LIN {X 0,Y 171.052,Z 952.165,A -85,B 0,C 180,E1 8008.321,E2 8008.321} C_VEL
LIN {X 0,Y 174.911,Z 942.549,A -85,B 0,C 180,E1 8004.093,E2 8004.093} C_VEL
LIN {X 0,Y 179.129,Z 931.53,A -85,B 0,C 180,E1 8000.36,E2 8000.36} C_VEL
LIN {X 0,Y 183.775,Z 918.134,A -85,B 0,C 180,E1 7996.88,E2 7996.88} C_VEL
LIN {X 0,Y 187.844,Z 904.879,A -85,B 0,C 180,E1 7994.248,E2 7994.248} C_VEL
LIN {X 0,Y 191.799,Z 889.443,A -85,B 0,C 180,E1 7991.93,E2 7991.93} C_VEL
LIN {X 0,Y 194.927,Z 873.983,A -85,B 0,C 180,E1 7990.211,E2 7990.211} C_VEL
LIN {X 0,Y 197.39,Z 856.631,A -85,B 0,C 180,E1 7988.872,E2 7988.872} C_VEL
LIN {X 0,Y 198.822,Z 839.35,A -85,B 0,C 180,E1 7988.05,E2 7988.05} C_VEL
LIN {X 0,Y 203.826,Z 763.58,A -85,B 0,C 180,E1 7985.576,E2 7985.576} C_VEL
LIN {X 0,Y 200.047,Z 723.867,A -85,B 0,C 180,E1 7982.552,E2 7982.552} C_VEL
LIN {X 0,Y 192.576,Z 708.428,A -85,B 0,C 180,E1 7979.398,E2 7979.398} C_VEL
LIN {X 0,Y 189.739,Z 703.046,A -85,B 0,C 180,E1 7978.041,E2 7978.041} C_VEL
LIN {X 0,Y 187.484,Z 693.288,A -85,B 0,C 180,E1 7973.127,E2 7973.127} C_VEL
LIN {X 0,Y 185.114,Z 684.758,A -85,B 0,C 180,E1 7967.95,E2 7967.95} C_VEL
LIN {X 0,Y 182.975,Z 677.799,A -85,B 0,C 180,E1 7962.924,E2 7962.924} C_VEL
LIN {X 0,Y 180.958,Z 671.792,A -85,B 0,C 180,E1 7957.631,E2 7957.631} C_VEL
LIN {X 0,Y 179.391,Z 667.819,A -85,B 0,C 180,E1 7953.109,E2 7953.109} C_VEL
LIN {X 0,Y 178.095,Z 664.338,A -85,B 0,C 180,E1 7948.138,E2 7948.138} C_VEL
LIN {X 0,Y 176.788,Z 660.79,A -85,B 0,C 180,E1 7939.838,E2 7939.838} C_VEL
LIN {X 0,Y 176.356,Z 660.229,A -85,B 0,C 180,E1 7933.442,E2 7933.442} C_VEL
LIN {X 0,Y 176.924,Z 660.85,A -85,B 0,C 180,E1 7927.143,E2 7927.143} C_VEL
LIN {X 0,Y 177.553,Z 662.846,A -85,B 0,C 180,E1 7922.26,E2 7922.26} C_VEL
LIN {X 0,Y 179.139,Z 665.796,A -85,B 0,C 180,E1 7916.801,E2 7916.801} C_VEL
LIN {X 0,Y 180.896,Z 669.96,A -85,B 0,C 180,E1 7911.738,E2 7911.738} C_VEL
LIN {X 0,Y 182.615,Z 674.195,A -85,B 0,C 180,E1 7907.671,E2 7907.671} C_VEL
LIN {X 0,Y 185.129,Z 680.488,A -85,B 0,C 180,E1 7902.72,E2 7902.72} C_VEL
LIN {X 0,Y 188.226,Z 689.312,A -85,B 0,C 180,E1 7897.184,E2 7897.184} C_VEL
LIN {X 0,Y 191.226,Z 698.648,A -85,B 0,C 180,E1 7892.416,E2 7892.416} C_VEL
LIN {X 0,Y 199.887,Z 713.757,A -85,B 0,C 180,E1 7888.779,E2 7888.779} C_VEL
LIN {X 0,Y 208.278,Z 730.588,A -85,B 0,C 180,E1 7885.621,E2 7885.621} C_VEL
LIN {X 0,Y 209.07,Z 733.001,A -85,B 0,C 180,E1 7885.302,E2 7885.302} C_VEL
LIN {X 0,Y 209.295,Z 744.68,A -85,B 0,C 180,E1 7884.7,E2 7884.7} C_VEL
LIN {X 0,Y 204.046,Z 825.384,A -85,B 0,C 180,E1 7882.3,E2 7882.3} C_VEL
LIN {X 0,Y 202.813,Z 833.052,A -85,B 0,C 180,E1 7882.253,E2 7882.253} C_VEL
LIN {X 0,Y 196.734,Z 853.33,A -85,B 0,C 180,E1 7882.805,E2 7882.805} C_VEL
LIN {X 0,Y 195.772,Z 859.913,A -85,B 0,C 180,E1 7882.739,E2 7882.739} C_VEL
LIN {X 0,Y 194.086,Z 879.533,A -85,B 0,C 180,E1 7881.974,E2 7881.974} C_VEL
LIN {X 0,Y 191.393,Z 896.772,A -85,B 0,C 180,E1 7880.877,E2 7880.877} C_VEL
LIN {X 0,Y 187.689,Z 913.328,A -85,B 0,C 180,E1 7879.389,E2 7879.389} C_VEL
LIN {X 0,Y 183.008,Z 930.142,A -85,B 0,C 180,E1 7877.295,E2 7877.295} C_VEL
LIN {X 0,Y 177.846,Z 945.933,A -85,B 0,C 180,E1 7874.65,E2 7874.65} C_VEL
LIN {X 0,Y 172.438,Z 960.631,A -85,B 0,C 180,E1 7871.378,E2 7871.378} C_VEL
LIN {X 0,Y 167.021,Z 974.241,A -85,B 0,C 180,E1 7867.419,E2 7867.419} C_VEL
LIN {X 0,Y 162.202,Z 986.322,A -85,B 0,C 180,E1 7862.852,E2 7862.852} C_VEL
LIN {X 0,Y 158.332,Z 996.58,A -85,B 0,C 180,E1 7857.861,E2 7857.861} C_VEL
LIN {X 0,Y 155.474,Z 1005.619,A -85,B 0,C 180,E1 7852.171,E2 7852.171} C_VEL
LIN {X 0,Y 154.031,Z 1012.929,A -85,B 0,C 180,E1 7846.116,E2 7846.116} C_VEL
LIN {X 0,Y 154.049,Z 1018.633,A -85,B 0,C 180,E1 7839.716,E2 7839.716} C_VEL
LIN {X 0,Y 155.156,Z 1022.277,A -85,B 0,C 180,E1 7833.696,E2 7833.696} C_VEL
LIN {X 0,Y 155.745,Z 1023.623,A -85,B 0,C 180,E1 7830.001,E2 7830.001} C_VEL
LIN {X 0,Y 154.747,Z 1024.067,A -85,B 0,C 180,E1 7825.554,E2 7825.554} C_VEL
LIN {X 0,Y 153.525,Z 1023.151,A -85,B 0,C 180,E1 7819.114,E2 7819.114} C_VEL
LIN {X 0,Y 153.864,Z 1020.428,A -85,B 0,C 180,E1 7812.217,E2 7812.217} C_VEL
LIN {X 0,Y 156.454,Z 1015.626,A -85,B 0,C 180,E1 7805.053,E2 7805.053} C_VEL
LIN {X 0,Y 161.104,Z 1009.155,A -85,B 0,C 180,E1 7798.579,E2 7798.579} C_VEL
LIN {X 0,Y 167.354,Z 1001.09,A -85,B 0,C 180,E1 7792.885,E2 7792.885} C_VEL
LIN {X 0,Y 174.735,Z 991.559,A -85,B 0,C 180,E1 7787.973,E2 7787.973} C_VEL
LIN {X 0,Y 182.872,Z 980.59,A -85,B 0,C 180,E1 7783.804,E2 7783.804} C_VEL
LIN {X 0,Y 191.37,Z 968.139,A -85,B 0,C 180,E1 7780.288,E2 7780.288} C_VEL
LIN {X 0,Y 199.606,Z 954.564,A -85,B 0,C 180,E1 7777.444,E2 7777.444} C_VEL
LIN {X 0,Y 207.323,Z 939.977,A -85,B 0,C 180,E1 7775.17,E2 7775.17} C_VEL
LIN {X 0,Y 214.323,Z 924.465,A -85,B 0,C 180,E1 7773.377,E2 7773.377} C_VEL
LIN {X 0,Y 220.444,Z 907.954,A -85,B 0,C 180,E1 7771.987,E2 7771.987} C_VEL
LIN {X 0,Y 225.279,Z 890.795,A -85,B 0,C 180,E1 7770.956,E2 7770.956} C_VEL
LIN {X 0,Y 228.713,Z 872.873,A -85,B 0,C 180,E1 7770.206,E2 7770.206} C_VEL
LIN {X 0,Y 231.397,Z 846.525,A -85,B 0,C 180,E1 7769.481,E2 7769.481} C_VEL
LIN {X 0,Y 238.924,Z 762.658,A -85,B 0,C 180,E1 7767.341,E2 7767.341} C_VEL
LIN {X 0,Y 234.578,Z 754.168,A -85,B 0,C 180,E1 7764.153,E2 7764.153} C_VEL
LIN {X 0,Y 231.17,Z 748.178,A -85,B 0,C 180,E1 7761.171,E2 7761.171} C_VEL
LIN {X 0,Y 228.461,Z 743.864,A -85,B 0,C 180,E1 7758.367,E2 7758.367} C_VEL
LIN {X 0,Y 225.969,Z 740.04,A -85,B 0,C 180,E1 7755.001,E2 7755.001} C_VEL
LIN {X 0,Y 223.932,Z 737.117,A -85,B 0,C 180,E1 7751.069,E2 7751.069} C_VEL
LIN {X 0,Y 222.678,Z 736.115,A -85,B 0,C 180,E1 7745.669,E2 7745.669} C_VEL
LIN {X 0,Y 222.804,Z 736.608,A -85,B 0,C 180,E1 7742.572,E2 7742.572} C_VEL
LIN {X 0,Y 224.405,Z 740.091,A -85,B 0,C 180,E1 7737.062,E2 7737.062} C_VEL
LIN {X 0,Y 226.766,Z 744.94,A -85,B 0,C 180,E1 7733.035,E2 7733.035} C_VEL
LIN {X 0,Y 228.583,Z 748.757,A -85,B 0,C 180,E1 7730.686,E2 7730.686} C_VEL
LIN {X 0,Y 231.247,Z 754.355,A -85,B 0,C 180,E1 7727.894,E2 7727.894} C_VEL
LIN {X 0,Y 234.202,Z 761.168,A -85,B 0,C 180,E1 7725.221,E2 7725.221} C_VEL
LIN {X 0,Y 235.779,Z 765.509,A -85,B 0,C 180,E1 7723.904,E2 7723.904} C_VEL
LIN {X 0,Y 236.085,Z 777.578,A -85,B 0,C 180,E1 7722.777,E2 7722.777} C_VEL
LIN {X 0,Y 228.922,Z 852.059,A -85,B 0,C 180,E1 7720.74,E2 7720.74} C_VEL
LIN {X 0,Y 226.241,Z 868.551,A -85,B 0,C 180,E1 7719.928,E2 7719.928} C_VEL
LIN {X 0,Y 222.3,Z 884.631,A -85,B 0,C 180,E1 7718.775,E2 7718.775} C_VEL
LIN {X 0,Y 217.471,Z 899.315,A -85,B 0,C 180,E1 7717.34,E2 7717.34} C_VEL
LIN {X 0,Y 211.583,Z 913.363,A -85,B 0,C 180,E1 7715.509,E2 7715.509} C_VEL
LIN {X 0,Y 204.895,Z 926.51,A -85,B 0,C 180,E1 7713.254,E2 7713.254} C_VEL
LIN {X 0,Y 197.577,Z 938.587,A -85,B 0,C 180,E1 7710.507,E2 7710.507} C_VEL
LIN {X 0,Y 190.099,Z 949.092,A -85,B 0,C 180,E1 7707.304,E2 7707.304} C_VEL
LIN {X 0,Y 182.682,Z 958.18,A -85,B 0,C 180,E1 7703.568,E2 7703.568} C_VEL
LIN {X 0,Y 175.545,Z 965.705,A -85,B 0,C 180,E1 7699.247,E2 7699.247} C_VEL
LIN {X 0,Y 169.015,Z 971.648,A -85,B 0,C 180,E1 7694.271,E2 7694.271} C_VEL
LIN {X 0,Y 163.752,Z 975.649,A -85,B 0,C 180,E1 7688.969,E2 7688.969} C_VEL
LIN {X 0,Y 159.527,Z 977.967,A -85,B 0,C 180,E1 7682.873,E2 7682.873} C_VEL
LIN {X 0,Y 157.008,Z 978.38,A -85,B 0,C 180,E1 7676.881,E2 7676.881} C_VEL
LIN {X 0,Y 155.83,Z 976.96,A -85,B 0,C 180,E1 7670.664,E2 7670.664} C_VEL
LIN {X 0,Y 155.953,Z 973.799,A -85,B 0,C 180,E1 7664.479,E2 7664.479} C_VEL
LIN {X 0,Y 157.211,Z 969.095,A -85,B 0,C 180,E1 7658.779,E2 7658.779} C_VEL
LIN {X 0,Y 159.818,Z 962.101,A -85,B 0,C 180,E1 7652.868,E2 7652.868} C_VEL
LIN {X 0,Y 163.179,Z 954.027,A -85,B 0,C 180,E1 7647.892,E2 7647.892} C_VEL
LIN {X 0,Y 167.51,Z 943.761,A -85,B 0,C 180,E1 7643.143,E2 7643.143} C_VEL
LIN {X 0,Y 172.022,Z 932.571,A -85,B 0,C 180,E1 7639.206,E2 7639.206} C_VEL
LIN {X 0,Y 176.924,Z 919.114,A -85,B 0,C 180,E1 7635.601,E2 7635.601} C_VEL
LIN {X 0,Y 181.29,Z 905.521,A -85,B 0,C 180,E1 7632.838,E2 7632.838} C_VEL
LIN {X 0,Y 185.432,Z 890.034,A -85,B 0,C 180,E1 7630.469,E2 7630.469} C_VEL
LIN {X 0,Y 188.703,Z 874.498,A -85,B 0,C 180,E1 7628.718,E2 7628.718} C_VEL
LIN {X 0,Y 191.28,Z 857.063,A -85,B 0,C 180,E1 7627.355,E2 7627.355} C_VEL
LIN {X 0,Y 192.774,Z 839.697,A -85,B 0,C 180,E1 7626.521,E2 7626.521} C_VEL
LIN {X 0,Y 197.948,Z 764.66,A -85,B 0,C 180,E1 7624.041,E2 7624.041} C_VEL
LIN {X 0,Y 194.607,Z 727.355,A -85,B 0,C 180,E1 7621.099,E2 7621.099} C_VEL
LIN {X 0,Y 187.847,Z 713.204,A -85,B 0,C 180,E1 7618.03,E2 7618.03} C_VEL
LIN {X 0,Y 182.177,Z 702.449,A -85,B 0,C 180,E1 7615.069,E2 7615.069} C_VEL
LIN {X 0,Y 180.219,Z 694.162,A -85,B 0,C 180,E1 7610.355,E2 7610.355} C_VEL
LIN {X 0,Y 178.087,Z 686.232,A -85,B 0,C 180,E1 7604.973,E2 7604.973} C_VEL
LIN {X 0,Y 176.156,Z 680.092,A -85,B 0,C 180,E1 7599.896,E2 7599.896} C_VEL
LIN {X 0,Y 174.811,Z 676.385,A -85,B 0,C 180,E1 7596.096,E2 7596.096} C_VEL
LIN {X 0,Y 173.854,Z 673.503,A -85,B 0,C 180,E1 7592.726,E2 7592.726} C_VEL
LIN {X 0,Y 172.738,Z 670.26,A -85,B 0,C 180,E1 7587.961,E2 7587.961} C_VEL
LIN {X 0,Y 171.591,Z 666.868,A -85,B 0,C 180,E1 7579.754,E2 7579.754} C_VEL
LIN {X 0,Y 171.207,Z 666.35,A -85,B 0,C 180,E1 7573.51,E2 7573.51} C_VEL
LIN {X 0,Y 171.807,Z 667.008,A -85,B 0,C 180,E1 7567.021,E2 7567.021} C_VEL
LIN {X 0,Y 172.724,Z 669.754,A -85,B 0,C 180,E1 7560.664,E2 7560.664} C_VEL
LIN {X 0,Y 173.824,Z 671.76,A -85,B 0,C 180,E1 7557.033,E2 7557.033} C_VEL
LIN {X 0,Y 175.425,Z 675.669,A -85,B 0,C 180,E1 7552.138,E2 7552.138} C_VEL
LIN {X 0,Y 177.084,Z 679.948,A -85,B 0,C 180,E1 7547.942,E2 7547.942} C_VEL
LIN {X 0,Y 179.367,Z 685.878,A -85,B 0,C 180,E1 7543.151,E2 7543.151} C_VEL
LIN {X 0,Y 182.17,Z 694.216,A -85,B 0,C 180,E1 7537.747,E2 7537.747} C_VEL
LIN {X 0,Y 183.8,Z 699.123,A -85,B 0,C 180,E1 7535.151,E2 7535.151} C_VEL
LIN {X 0,Y 190.764,Z 710.817,A -85,B 0,C 180,E1 7531.855,E2 7531.855} C_VEL
LIN {X 0,Y 198.07,Z 724.565,A -85,B 0,C 180,E1 7528.757,E2 7528.757} C_VEL
LIN {X 0,Y 203.297,Z 735.747,A -85,B 0,C 180,E1 7526.702,E2 7526.702} C_VEL
LIN {X 0,Y 203.404,Z 745.5,A -85,B 0,C 180,E1 7526.197,E2 7526.197} C_VEL
LIN {X 0,Y 195.772,Z 859.913,A -85,B 0,C 180,E1 7522.739,E2 7522.739} C_VEL
LIN {X 0,Y 194.472,Z 867.56,A -85,B 0,C 180,E1 7522.678,E2 7522.678} C_VEL
LIN {X 0,Y 188.765,Z 883.336,A -85,B 0,C 180,E1 7522.945,E2 7522.945} C_VEL
LIN {X 0,Y 186.35,Z 890.745,A -85,B 0,C 180,E1 7522.781,E2 7522.781} C_VEL
LIN {X 0,Y 185.647,Z 893.958,A -85,B 0,C 180,E1 7522.594,E2 7522.594} C_VEL
LIN {X 0,Y 181.904,Z 910.745,A -85,B 0,C 180,E1 7521.129,E2 7521.129} C_VEL
LIN {X 0,Y 177.222,Z 927.25,A -85,B 0,C 180,E1 7519.115,E2 7519.115} C_VEL
LIN {X 0,Y 171.795,Z 943.419,A -85,B 0,C 180,E1 7516.437,E2 7516.437} C_VEL
LIN {X 0,Y 166.096,Z 958.432,A -85,B 0,C 180,E1 7513.118,E2 7513.118} C_VEL
LIN {X 0,Y 160.537,Z 971.798,A -85,B 0,C 180,E1 7509.211,E2 7509.211} C_VEL
LIN {X 0,Y 155.317,Z 984.104,A -85,B 0,C 180,E1 7504.508,E2 7504.508} C_VEL
LIN {X 0,Y 151.081,Z 994.558,A -85,B 0,C 180,E1 7499.324,E2 7499.324} C_VEL
LIN {X 0,Y 147.934,Z 1003.622,A -85,B 0,C 180,E1 7493.502,E2 7493.502} C_VEL
LIN {X 0,Y 146.187,Z 1011.195,A -85,B 0,C 180,E1 7487.105,E2 7487.105} C_VEL
LIN {X 0,Y 146.016,Z 1016.842,A -85,B 0,C 180,E1 7480.655,E2 7480.655} C_VEL
LIN {X 0,Y 147.075,Z 1020.719,A -85,B 0,C 180,E1 7474.289,E2 7474.289} C_VEL
LIN {X 0,Y 147.827,Z 1022.202,A -85,B 0,C 180,E1 7470.388,E2 7470.388} C_VEL
LIN {X 0,Y 147.171,Z 1022.745,A -85,B 0,C 180,E1 7466.885,E2 7466.885} C_VEL
LIN {X 0,Y 145.694,Z 1022.297,A -85,B 0,C 180,E1 7460.122,E2 7460.122} C_VEL
LIN {X 0,Y 145.776,Z 1020.07,A -85,B 0,C 180,E1 7452.847,E2 7452.847} C_VEL
LIN {X 0,Y 148.008,Z 1016.078,A -85,B 0,C 180,E1 7445.665,E2 7445.665} C_VEL
LIN {X 0,Y 152.508,Z 1010.2,A -85,B 0,C 180,E1 7438.807,E2 7438.807} C_VEL
LIN {X 0,Y 158.718,Z 1002.814,A -85,B 0,C 180,E1 7432.789,E2 7432.789} C_VEL
LIN {X 0,Y 166.649,Z 993.414,A -85,B 0,C 180,E1 7427.315,E2 7427.315} C_VEL
LIN {X 0,Y 174.937,Z 983.139,A -85,B 0,C 180,E1 7422.981,E2 7422.981} C_VEL
LIN {X 0,Y 183.602,Z 971.42,A -85,B 0,C 180,E1 7419.349,E2 7419.349} C_VEL
LIN {X 0,Y 192.339,Z 958.228,A -85,B 0,C 180,E1 7416.317,E2 7416.317} C_VEL
LIN {X 0,Y 200.577,Z 944.065,A -85,B 0,C 180,E1 7413.903,E2 7413.903} C_VEL
LIN {X 0,Y 207.918,Z 929.335,A -85,B 0,C 180,E1 7412.043,E2 7412.043} C_VEL
LIN {X 0,Y 214.334,Z 913.885,A -85,B 0,C 180,E1 7410.607,E2 7410.607} C_VEL
LIN {X 0,Y 219.711,Z 897.447,A -85,B 0,C 180,E1 7409.502,E2 7409.502} C_VEL
LIN {X 0,Y 223.895,Z 879.754,A -85,B 0,C 180,E1 7408.656,E2 7408.656} C_VEL
LIN {X 0,Y 226.524,Z 861.629,A -85,B 0,C 180,E1 7408.063,E2 7408.063} C_VEL
LIN {X 0,Y 235.316,Z 767.051,A -85,B 0,C 180,E1 7405.683,E2 7405.683} C_VEL
LIN {X 0,Y 231.684,Z 759.881,A -85,B 0,C 180,E1 7402.721,E2 7402.721} C_VEL
LIN {X 0,Y 229.265,Z 755.373,A -85,B 0,C 180,E1 7400.419,E2 7400.419} C_VEL
LIN {X 0,Y 226.828,Z 751.284,A -85,B 0,C 180,E1 7397.707,E2 7397.707} C_VEL
LIN {X 0,Y 224.564,Z 747.63,A -85,B 0,C 180,E1 7394.438,E2 7394.438} C_VEL
LIN {X 0,Y 222.827,Z 745.003,A -85,B 0,C 180,E1 7390.862,E2 7390.862} C_VEL
LIN {X 0,Y 221.647,Z 744.048,A -85,B 0,C 180,E1 7385.435,E2 7385.435} C_VEL
LIN {X 0,Y 221.776,Z 744.618,A -85,B 0,C 180,E1 7382.583,E2 7382.583} C_VEL
LIN {X 0,Y 223.198,Z 747.898,A -85,B 0,C 180,E1 7377.397,E2 7377.397} C_VEL
LIN {X 0,Y 225.684,Z 753.33,A -85,B 0,C 180,E1 7373.001,E2 7373.001} C_VEL
LIN {X 0,Y 229.024,Z 760.874,A -85,B 0,C 180,E1 7368.925,E2 7368.925} C_VEL
LIN {X 0,Y 231.924,Z 767.971,A -85,B 0,C 180,E1 7366.092,E2 7366.092} C_VEL
LIN {X 0,Y 232.709,Z 770.494,A -85,B 0,C 180,E1 7365.347,E2 7365.347} C_VEL
LIN {X 0,Y 232.775,Z 779.251,A -85,B 0,C 180,E1 7364.536,E2 7364.536} C_VEL
LIN {X 0,Y 225.455,Z 852.798,A -85,B 0,C 180,E1 7362.549,E2 7362.549} C_VEL
LIN {X 0,Y 222.635,Z 869.466,A -85,B 0,C 180,E1 7361.737,E2 7361.737} C_VEL
LIN {X 0,Y 218.42,Z 885.963,A -85,B 0,C 180,E1 7360.561,E2 7360.561} C_VEL
LIN {X 0,Y 213.383,Z 900.585,A -85,B 0,C 180,E1 7359.137,E2 7359.137} C_VEL
LIN {X 0,Y 207.066,Z 914.99,A -85,B 0,C 180,E1 7357.261,E2 7357.261} C_VEL
LIN {X 0,Y 199.819,Z 928.551,A -85,B 0,C 180,E1 7354.916,E2 7354.916} C_VEL
LIN {X 0,Y 192.206,Z 940.381,A -85,B 0,C 180,E1 7352.17,E2 7352.17} C_VEL
LIN {X 0,Y 184.405,Z 950.759,A -85,B 0,C 180,E1 7348.946,E2 7348.946} C_VEL
LIN {X 0,Y 176.504,Z 959.852,A -85,B 0,C 180,E1 7345.099,E2 7345.099} C_VEL
LIN {X 0,Y 169.077,Z 967.149,A -85,B 0,C 180,E1 7340.745,E2 7340.745} C_VEL
LIN {X 0,Y 162.181,Z 972.997,A -85,B 0,C 180,E1 7335.655,E2 7335.655} C_VEL
LIN {X 0,Y 156.554,Z 976.935,A -85,B 0,C 180,E1 7330.169,E2 7330.169} C_VEL
LIN {X 0,Y 152.089,Z 979.18,A -85,B 0,C 180,E1 7323.973,E2 7323.973} C_VEL
LIN {X 0,Y 149.246,Z 979.592,A -85,B 0,C 180,E1 7317.532,E2 7317.532} C_VEL
LIN {X 0,Y 147.929,Z 978.145,A -85,B 0,C 180,E1 7310.991,E2 7310.991} C_VEL
LIN {X 0,Y 148.015,Z 974.962,A -85,B 0,C 180,E1 7304.473,E2 7304.473} C_VEL
LIN {X 0,Y 149.321,Z 970.243,A -85,B 0,C 180,E1 7298.471,E2 7298.471} C_VEL
LIN {X 0,Y 152.061,Z 963.242,A -85,B 0,C 180,E1 7292.26,E2 7292.26} C_VEL
LIN {X 0,Y 155.599,Z 955.176,A -85,B 0,C 180,E1 7287.053,E2 7287.053} C_VEL
LIN {X 0,Y 160.155,Z 944.923,A -85,B 0,C 180,E1 7282.105,E2 7282.105} C_VEL
LIN {X 0,Y 164.918,Z 933.712,A -85,B 0,C 180,E1 7278.004,E2 7278.004} C_VEL
LIN {X 0,Y 170.031,Z 920.363,A -85,B 0,C 180,E1 7274.305,E2 7274.305} C_VEL
LIN {X 0,Y 174.597,Z 906.881,A -85,B 0,C 180,E1 7271.467,E2 7271.467} C_VEL
LIN {X 0,Y 178.924,Z 891.513,A -85,B 0,C 180,E1 7269.044,E2 7269.044} C_VEL
LIN {X 0,Y 182.344,Z 876.263,A -85,B 0,C 180,E1 7267.258,E2 7267.258} C_VEL
LIN {X 0,Y 185.04,Z 859.26,A -85,B 0,C 180,E1 7265.869,E2 7265.869} C_VEL
LIN {X 0,Y 186.703,Z 842.012,A -85,B 0,C 180,E1 7264.981,E2 7264.981} C_VEL
LIN {X 0,Y 192.17,Z 765.586,A -85,B 0,C 180,E1 7262.414,E2 7262.414} C_VEL
LIN {X 0,Y 189.372,Z 731.111,A -85,B 0,C 180,E1 7259.603,E2 7259.603} C_VEL
LIN {X 0,Y 183.39,Z 718.266,A -85,B 0,C 180,E1 7256.673,E2 7256.673} C_VEL
LIN {X 0,Y 177.15,Z 706.691,A -85,B 0,C 180,E1 7253.34,E2 7253.34} C_VEL
LIN {X 0,Y 174.863,Z 702.316,A -85,B 0,C 180,E1 7251.862,E2 7251.862} C_VEL
LIN {X 0,Y 172.859,Z 694.084,A -85,B 0,C 180,E1 7246.501,E2 7246.501} C_VEL
LIN {X 0,Y 170.992,Z 687.629,A -85,B 0,C 180,E1 7241.359,E2 7241.359} C_VEL
LIN {X 0,Y 169.52,Z 682.678,A -85,B 0,C 180,E1 7236.565,E2 7236.565} C_VEL
LIN {X 0,Y 168.332,Z 679.192,A -85,B 0,C 180,E1 7232.316,E2 7232.316} C_VEL
LIN {X 0,Y 167.397,Z 676.194,A -85,B 0,C 180,E1 7227.769,E2 7227.769} C_VEL
LIN {X 0,Y 166.359,Z 672.888,A -85,B 0,C 180,E1 7219.304,E2 7219.304} C_VEL
LIN {X 0,Y 166.079,Z 672.48,A -85,B 0,C 180,E1 7212.756,E2 7212.756} C_VEL
LIN {X 0,Y 166.746,Z 673.248,A -85,B 0,C 180,E1 7206.543,E2 7206.543} C_VEL
LIN {X 0,Y 168.453,Z 677.442,A -85,B 0,C 180,E1 7197.619,E2 7197.619} C_VEL
LIN {X 0,Y 170.043,Z 681.719,A -85,B 0,C 180,E1 7192.228,E2 7192.228} C_VEL
LIN {X 0,Y 171.541,Z 685.68,A -85,B 0,C 180,E1 7188.229,E2 7188.229} C_VEL
LIN {X 0,Y 173.724,Z 691.718,A -85,B 0,C 180,E1 7183.276,E2 7183.276} C_VEL
LIN {X 0,Y 176.23,Z 699.176,A -85,B 0,C 180,E1 7178.404,E2 7178.404} C_VEL
LIN {X 0,Y 183.456,Z 710.887,A -85,B 0,C 180,E1 7174.541,E2 7174.541} C_VEL
LIN {X 0,Y 190.952,Z 724.711,A -85,B 0,C 180,E1 7171.001,E2 7171.001} C_VEL
LIN {X 0,Y 197.611,Z 738.73,A -85,B 0,C 180,E1 7168.155,E2 7168.155} C_VEL
LIN {X 0,Y 197.592,Z 746.541,A -85,B 0,C 180,E1 7167.76,E2 7167.76} C_VEL
LIN {X 0,Y 188.693,Z 872.713,A -85,B 0,C 180,E1 7163.829,E2 7163.829} C_VEL
LIN {X 0,Y 186.194,Z 890.837,A -85,B 0,C 180,E1 7162.808,E2 7162.808} C_VEL
LIN {X 0,Y 185.647,Z 893.958,A -85,B 0,C 180,E1 7162.594,E2 7162.594} C_VEL
LIN {X 0,Y 183.422,Z 901.307,A -85,B 0,C 180,E1 7162.228,E2 7162.228} C_VEL
LIN {X 0,Y 176.159,Z 915.134,A -85,B 0,C 180,E1 7161.787,E2 7161.787} C_VEL
LIN {X 0,Y 172.207,Z 922.932,A -85,B 0,C 180,E1 7161.192,E2 7161.192} C_VEL
LIN {X 0,Y 171.093,Z 925.859,A -85,B 0,C 180,E1 7160.816,E2 7160.816} C_VEL
LIN {X 0,Y 165.637,Z 941.563,A -85,B 0,C 180,E1 7158.204,E2 7158.204} C_VEL
LIN {X 0,Y 159.88,Z 956.17,A -85,B 0,C 180,E1 7154.967,E2 7154.967} C_VEL
LIN {X 0,Y 153.993,Z 969.81,A -85,B 0,C 180,E1 7150.98,E2 7150.98} C_VEL
LIN {X 0,Y 148.57,Z 981.875,A -85,B 0,C 180,E1 7146.317,E2 7146.317} C_VEL
LIN {X 0,Y 143.935,Z 992.534,A -85,B 0,C 180,E1 7140.935,E2 7140.935} C_VEL
LIN {X 0,Y 140.421,Z 1001.768,A -85,B 0,C 180,E1 7134.842,E2 7134.842} C_VEL
LIN {X 0,Y 138.367,Z 1009.518,A -85,B 0,C 180,E1 7128.104,E2 7128.104} C_VEL
LIN {X 0,Y 138.027,Z 1015.33,A -85,B 0,C 180,E1 7121.28,E2 7121.28} C_VEL
LIN {X 0,Y 139.065,Z 1019.331,A -85,B 0,C 180,E1 7114.537,E2 7114.537} C_VEL
LIN {X 0,Y 139.951,Z 1020.991,A -85,B 0,C 180,E1 7110.001,E2 7110.001} C_VEL
LIN {X 0,Y 138.839,Z 1021.534,A -85,B 0,C 180,E1 7105.457,E2 7105.457} C_VEL
LIN {X 0,Y 137.564,Z 1020.792,A -85,B 0,C 180,E1 7097.833,E2 7097.833} C_VEL
LIN {X 0,Y 138.382,Z 1018.128,A -85,B 0,C 180,E1 7089.932,E2 7089.932} C_VEL
LIN {X 0,Y 141.71,Z 1013.603,A -85,B 0,C 180,E1 7082.247,E2 7082.247} C_VEL
LIN {X 0,Y 147.379,Z 1007.249,A -85,B 0,C 180,E1 7075.174,E2 7075.174} C_VEL
LIN {X 0,Y 154.678,Z 999.394,A -85,B 0,C 180,E1 7069.139,E2 7069.139} C_VEL
LIN {X 0,Y 162.947,Z 990.157,A -85,B 0,C 180,E1 7064.117,E2 7064.117} C_VEL
LIN {X 0,Y 171.996,Z 979.401,A -85,B 0,C 180,E1 7059.884,E2 7059.884} C_VEL
LIN {X 0,Y 181.296,Z 967.19,A -85,B 0,C 180,E1 7056.371,E2 7056.371} C_VEL
LIN {X 0,Y 190.215,Z 953.969,A -85,B 0,C 180,E1 7053.577,E2 7053.577} C_VEL
LIN {X 0,Y 198.636,Z 939.481,A -85,B 0,C 180,E1 7051.336,E2 7051.336} C_VEL
LIN {X 0,Y 206.339,Z 923.717,A -85,B 0,C 180,E1 7049.564,E2 7049.564} C_VEL
LIN {X 0,Y 212.817,Z 907.457,A -85,B 0,C 180,E1 7048.248,E2 7048.248} C_VEL
LIN {X 0,Y 217.947,Z 890.747,A -85,B 0,C 180,E1 7047.271,E2 7047.271} C_VEL
LIN {X 0,Y 221.681,Z 872.965,A -85,B 0,C 180,E1 7046.543,E2 7046.543} C_VEL
LIN {X 0,Y 224.401,Z 849.303,A -85,B 0,C 180,E1 7045.895,E2 7045.895} C_VEL
LIN {X 0,Y 231.925,Z 771.64,A -85,B 0,C 180,E1 7043.974,E2 7043.974} C_VEL
LIN {X 0,Y 228.415,Z 764.31,A -85,B 0,C 180,E1 7040.699,E2 7040.699} C_VEL
LIN {X 0,Y 225.321,Z 758.846,A -85,B 0,C 180,E1 7037.163,E2 7037.163} C_VEL
LIN {X 0,Y 223.179,Z 755.22,A -85,B 0,C 180,E1 7033.867,E2 7033.867} C_VEL
LIN {X 0,Y 221.628,Z 752.803,A -85,B 0,C 180,E1 7030.396,E2 7030.396} C_VEL
LIN {X 0,Y 220.608,Z 751.99,A -85,B 0,C 180,E1 7024.94,E2 7024.94} C_VEL
LIN {X 0,Y 220.743,Z 752.625,A -85,B 0,C 180,E1 7022.596,E2 7022.596} C_VEL
LIN {X 0,Y 221.961,Z 755.642,A -85,B 0,C 180,E1 7017.805,E2 7017.805} C_VEL
LIN {X 0,Y 224.594,Z 761.771,A -85,B 0,C 180,E1 7012.967,E2 7012.967} C_VEL
LIN {X 0,Y 227.251,Z 768.387,A -85,B 0,C 180,E1 7009.543,E2 7009.543} C_VEL
LIN {X 0,Y 229.807,Z 775.086,A -85,B 0,C 180,E1 7006.875,E2 7006.875} C_VEL
LIN {X 0,Y 229.753,Z 780.959,A -85,B 0,C 180,E1 7006.349,E2 7006.349} C_VEL
LIN {X 0,Y 222.277,Z 853.477,A -85,B 0,C 180,E1 7004.42,E2 7004.42} C_VEL
LIN {X 0,Y 219.355,Z 870.12,A -85,B 0,C 180,E1 7003.622,E2 7003.622} C_VEL
LIN {X 0,Y 214.962,Z 886.699,A -85,B 0,C 180,E1 7002.463,E2 7002.463} C_VEL
LIN {X 0,Y 209.859,Z 901.043,A -85,B 0,C 180,E1 7001.095,E2 7001.095} C_VEL
LIN {X 0,Y 203.191,Z 915.745,A -85,B 0,C 180,E1 6999.219,E2 6999.219} C_VEL
LIN {X 0,Y 195.653,Z 929.339,A -85,B 0,C 180,E1 6996.906,E2 6996.906} C_VEL
LIN {X 0,Y 187.709,Z 941.226,A -85,B 0,C 180,E1 6994.184,E2 6994.184} C_VEL
LIN {X 0,Y 179.527,Z 951.639,A -85,B 0,C 180,E1 6990.973,E2 6990.973} C_VEL
LIN {X 0,Y 171.144,Z 960.837,A -85,B 0,C 180,E1 6987.089,E2 6987.089} C_VEL
LIN {X 0,Y 163.232,Z 968.198,A -85,B 0,C 180,E1 6982.668,E2 6982.668} C_VEL
LIN {X 0,Y 155.902,Z 974.031,A -85,B 0,C 180,E1 6977.522,E2 6977.522} C_VEL
LIN {X 0,Y 149.793,Z 978.042,A -85,B 0,C 180,E1 6971.873,E2 6971.873} C_VEL
LIN {X 0,Y 144.863,Z 980.342,A -85,B 0,C 180,E1 6965.434,E2 6965.434} C_VEL
LIN {X 0,Y 141.649,Z 980.834,A -85,B 0,C 180,E1 6958.684,E2 6958.684} C_VEL
LIN {X 0,Y 140.081,Z 979.474,A -85,B 0,C 180,E1 6951.787,E2 6951.787} C_VEL
LIN {X 0,Y 140.029,Z 976.364,A -85,B 0,C 180,E1 6944.895,E2 6944.895} C_VEL
LIN {X 0,Y 141.306,Z 971.775,A -85,B 0,C 180,E1 6938.545,E2 6938.545} C_VEL
LIN {X 0,Y 143.879,Z 965.366,A -85,B 0,C 180,E1 6932.389,E2 6932.389} C_VEL
LIN {X 0,Y 147.454,Z 957.597,A -85,B 0,C 180,E1 6926.89,E2 6926.89} C_VEL
LIN {X 0,Y 151.745,Z 948.501,A -85,B 0,C 180,E1 6922.046,E2 6922.046} C_VEL
LIN {X 0,Y 156.886,Z 937.146,A -85,B 0,C 180,E1 6917.485,E2 6917.485} C_VEL
LIN {X 0,Y 162.044,Z 924.739,A -85,B 0,C 180,E1 6913.694,E2 6913.694} C_VEL
LIN {X 0,Y 167.227,Z 910.504,A -85,B 0,C 180,E1 6910.437,E2 6910.437} C_VEL
LIN {X 0,Y 171.728,Z 896.028,A -85,B 0,C 180,E1 6907.941,E2 6907.941} C_VEL
LIN {X 0,Y 175.582,Z 880.369,A -85,B 0,C 180,E1 6905.953,E2 6905.953} C_VEL
LIN {X 0,Y 178.657,Z 863.555,A -85,B 0,C 180,E1 6904.428,E2 6904.428} C_VEL
LIN {X 0,Y 180.615,Z 846.139,A -85,B 0,C 180,E1 6903.424,E2 6903.424} C_VEL
LIN {X 0,Y 186.568,Z 766.675,A -85,B 0,C 180,E1 6900.7,E2 6900.7} C_VEL
LIN {X 0,Y 184.157,Z 734.521,A -85,B 0,C 180,E1 6897.96,E2 6897.96} C_VEL
LIN {X 0,Y 177.846,Z 720.915,A -85,B 0,C 180,E1 6894.608,E2 6894.608} C_VEL
LIN {X 0,Y 172.577,Z 711.043,A -85,B 0,C 180,E1 6891.526,E2 6891.526} C_VEL
LIN {X 0,Y 167.675,Z 702.402,A -85,B 0,C 180,E1 6888.193,E2 6888.193} C_VEL
LIN {X 0,Y 165.92,Z 695.588,A -85,B 0,C 180,E1 6883.182,E2 6883.182} C_VEL
LIN {X 0,Y 164.351,Z 689.912,A -85,B 0,C 180,E1 6877.913,E2 6877.913} C_VEL
LIN {X 0,Y 162.937,Z 685.122,A -85,B 0,C 180,E1 6872.269,E2 6872.269} C_VEL
LIN {X 0,Y 161.961,Z 681.978,A -85,B 0,C 180,E1 6867.184,E2 6867.184} C_VEL
LIN {X 0,Y 161.16,Z 678.962,A -85,B 0,C 180,E1 6859.198,E2 6859.198} C_VEL
LIN {X 0,Y 160.944,Z 678.611,A -85,B 0,C 180,E1 6852.559,E2 6852.559} C_VEL
LIN {X 0,Y 161.596,Z 679.438,A -85,B 0,C 180,E1 6846.395,E2 6846.395} C_VEL
LIN {X 0,Y 163.185,Z 683.664,A -85,B 0,C 180,E1 6837.543,E2 6837.543} C_VEL
LIN {X 0,Y 164.576,Z 687.417,A -85,B 0,C 180,E1 6832.671,E2 6832.671} C_VEL
LIN {X 0,Y 165.995,Z 691.401,A -85,B 0,C 180,E1 6828.535,E2 6828.535} C_VEL
LIN {X 0,Y 168.09,Z 697.546,A -85,B 0,C 180,E1 6823.411,E2 6823.411} C_VEL
LIN {X 0,Y 169.115,Z 699.999,A -85,B 0,C 180,E1 6821.918,E2 6821.918} C_VEL
LIN {X 0,Y 173.935,Z 707.532,A -85,B 0,C 180,E1 6818.856,E2 6818.856} C_VEL
LIN {X 0,Y 179.573,Z 716.842,A -85,B 0,C 180,E1 6815.712,E2 6815.712} C_VEL
LIN {X 0,Y 186.697,Z 730.395,A -85,B 0,C 180,E1 6812.144,E2 6812.144} C_VEL
LIN {X 0,Y 192.076,Z 742.205,A -85,B 0,C 180,E1 6809.661,E2 6809.661} C_VEL
LIN {X 0,Y 191.761,Z 749.825,A -85,B 0,C 180,E1 6809.348,E2 6809.348} C_VEL
LIN {X 0,Y 182.744,Z 872.225,A -85,B 0,C 180,E1 6805.484,E2 6805.484} C_VEL
LIN {X 0,Y 180.132,Z 890.396,A -85,B 0,C 180,E1 6804.443,E2 6804.443} C_VEL
LIN {X 0,Y 176.449,Z 907.28,A -85,B 0,C 180,E1 6803.035,E2 6803.035} C_VEL
LIN {X 0,Y 171.945,Z 923.212,A -85,B 0,C 180,E1 6801.189,E2 6801.189} C_VEL
LIN {X 0,Y 171.093,Z 925.859,A -85,B 0,C 180,E1 6800.816,E2 6800.816} C_VEL
LIN {X 0,Y 168.02,Z 932.65,A -85,B 0,C 180,E1 6799.974,E2 6799.974} C_VEL
LIN {X 0,Y 159.399,Z 945.099,A -85,B 0,C 180,E1 6798.592,E2 6798.592} C_VEL
LIN {X 0,Y 154.839,Z 952.006,A -85,B 0,C 180,E1 6797.397,E2 6797.397} C_VEL
LIN {X 0,Y 153.558,Z 954.543,A -85,B 0,C 180,E1 6796.793,E2 6796.793} C_VEL
LIN {X 0,Y 147.367,Z 968.246,A -85,B 0,C 180,E1 6792.726,E2 6792.726} C_VEL
LIN {X 0,Y 141.582,Z 980.417,A -85,B 0,C 180,E1 6787.909,E2 6787.909} C_VEL
LIN {X 0,Y 136.604,Z 991.15,A -85,B 0,C 180,E1 6782.299,E2 6782.299} C_VEL
LIN {X 0,Y 132.784,Z 1000.449,A -85,B 0,C 180,E1 6775.897,E2 6775.897} C_VEL
LIN {X 0,Y 130.505,Z 1008.248,A -85,B 0,C 180,E1 6768.772,E2 6768.772} C_VEL
LIN {X 0,Y 130.068,Z 1014.1,A -85,B 0,C 180,E1 6761.53,E2 6761.53} C_VEL
LIN {X 0,Y 131.144,Z 1018.121,A -85,B 0,C 180,E1 6754.373,E2 6754.373} C_VEL
LIN {X 0,Y 132.051,Z 1019.674,A -85,B 0,C 180,E1 6750.001,E2 6750.001} C_VEL
LIN {X 0,Y 130.712,Z 1020.262,A -85,B 0,C 180,E1 6744.734,E2 6744.734} C_VEL
LIN {X 0,Y 129.603,Z 1019.501,A -85,B 0,C 180,E1 6736.619,E2 6736.619} C_VEL
LIN {X 0,Y 130.77,Z 1016.936,A -85,B 0,C 180,E1 6728.47,E2 6728.47} C_VEL
LIN {X 0,Y 134.706,Z 1012.362,A -85,B 0,C 180,E1 6720.276,E2 6720.276} C_VEL
LIN {X 0,Y 141.041,Z 1006.008,A -85,B 0,C 180,E1 6712.946,E2 6712.946} C_VEL
LIN {X 0,Y 148.973,Z 998.185,A -85,B 0,C 180,E1 6706.797,E2 6706.797} C_VEL
LIN {X 0,Y 158.134,Z 988.66,A -85,B 0,C 180,E1 6701.597,E2 6701.597} C_VEL
LIN {X 0,Y 168.235,Z 977.268,A -85,B 0,C 180,E1 6697.213,E2 6697.213} C_VEL
LIN {X 0,Y 178.055,Z 964.859,A -85,B 0,C 180,E1 6693.79,E2 6693.79} C_VEL
LIN {X 0,Y 187.398,Z 951.3,A -85,B 0,C 180,E1 6691.092,E2 6691.092} C_VEL
LIN {X 0,Y 195.971,Z 936.788,A -85,B 0,C 180,E1 6688.992,E2 6688.992} C_VEL
LIN {X 0,Y 203.743,Z 921.086,A -85,B 0,C 180,E1 6687.346,E2 6687.346} C_VEL
LIN {X 0,Y 209.994,Z 905.547,A -85,B 0,C 180,E1 6686.167,E2 6686.167} C_VEL
LIN {X 0,Y 215.226,Z 888.475,A -85,B 0,C 180,E1 6685.232,E2 6685.232} C_VEL
LIN {X 0,Y 218.946,Z 870.63,A -85,B 0,C 180,E1 6684.547,E2 6684.547} C_VEL
LIN {X 0,Y 221.997,Z 843.629,A -85,B 0,C 180,E1 6683.845,E2 6683.845} C_VEL
LIN {X 0,Y 228.767,Z 776.294,A -85,B 0,C 180,E1 6682.213,E2 6682.213} C_VEL
LIN {X 0,Y 225.802,Z 770.13,A -85,B 0,C 180,E1 6679.127,E2 6679.127} C_VEL
LIN {X 0,Y 223.654,Z 766.119,A -85,B 0,C 180,E1 6676.358,E2 6676.358} C_VEL
LIN {X 0,Y 221.816,Z 762.808,A -85,B 0,C 180,E1 6673.29,E2 6673.29} C_VEL
LIN {X 0,Y 220.528,Z 760.688,A -85,B 0,C 180,E1 6670.184,E2 6670.184} C_VEL
LIN {X 0,Y 219.587,Z 759.925,A -85,B 0,C 180,E1 6664.963,E2 6664.963} C_VEL
LIN {X 0,Y 219.709,Z 760.63,A -85,B 0,C 180,E1 6662.608,E2 6662.608} C_VEL
LIN {X 0,Y 220.812,Z 763.54,A -85,B 0,C 180,E1 6658.053,E2 6658.053} C_VEL
LIN {X 0,Y 223.114,Z 769.441,A -85,B 0,C 180,E1 6653.502,E2 6653.502} C_VEL
LIN {X 0,Y 225.403,Z 775.616,A -85,B 0,C 180,E1 6650.295,E2 6650.295} C_VEL
LIN {X 0,Y 227.072,Z 780.458,A -85,B 0,C 180,E1 6648.362,E2 6648.362} C_VEL
LIN {X 0,Y 226.854,Z 783.743,A -85,B 0,C 180,E1 6648.183,E2 6648.183} C_VEL
LIN {X 0,Y 219.358,Z 854.224,A -85,B 0,C 180,E1 6646.343,E2 6646.343} C_VEL
LIN {X 0,Y 216.311,Z 870.956,A -85,B 0,C 180,E1 6645.556,E2 6645.556} C_VEL
LIN {X 0,Y 211.753,Z 887.578,A -85,B 0,C 180,E1 6644.418,E2 6644.418} C_VEL
LIN {X 0,Y 206.421,Z 902.043,A -85,B 0,C 180,E1 6643.067,E2 6643.067} C_VEL
LIN {X 0,Y 199.568,Z 916.599,A -85,B 0,C 180,E1 6641.246,E2 6641.246} C_VEL
LIN {X 0,Y 191.738,Z 930.175,A -85,B 0,C 180,E1 6638.976,E2 6638.976} C_VEL
LIN {X 0,Y 183.457,Z 942.078,A -85,B 0,C 180,E1 6636.293,E2 6636.293} C_VEL
LIN {X 0,Y 174.199,Z 953.302,A -85,B 0,C 180,E1 6632.83,E2 6632.83} C_VEL
LIN {X 0,Y 165.612,Z 962.19,A -85,B 0,C 180,E1 6629.015,E2 6629.015} C_VEL
LIN {X 0,Y 157.198,Z 969.555,A -85,B 0,C 180,E1 6624.502,E2 6624.502} C_VEL
LIN {X 0,Y 149.321,Z 975.407,A -85,B 0,C 180,E1 6619.169,E2 6619.169} C_VEL
LIN {X 0,Y 142.665,Z 979.401,A -85,B 0,C 180,E1 6613.206,E2 6613.206} C_VEL
LIN {X 0,Y 137.191,Z 981.687,A -85,B 0,C 180,E1 6606.18,E2 6606.18} C_VEL
LIN {X 0,Y 133.767,Z 982.002,A -85,B 0,C 180,E1 6599.008,E2 6599.008} C_VEL
LIN {X 0,Y 132.095,Z 980.362,A -85,B 0,C 180,E1 6591.304,E2 6591.304} C_VEL
LIN {X 0,Y 132.143,Z 977.263,A -85,B 0,C 180,E1 6584.413,E2 6584.413} C_VEL
LIN {X 0,Y 133.555,Z 972.537,A -85,B 0,C 180,E1 6577.744,E2 6577.744} C_VEL
LIN {X 0,Y 136.606,Z 965.523,A -85,B 0,C 180,E1 6570.838,E2 6570.838} C_VEL
LIN {X 0,Y 140.556,Z 957.474,A -85,B 0,C 180,E1 6565.102,E2 6565.102} C_VEL
LIN {X 0,Y 145.625,Z 947.245,A -85,B 0,C 180,E1 6559.716,E2 6559.716} C_VEL
LIN {X 0,Y 150.93,Z 936.061,A -85,B 0,C 180,E1 6555.288,E2 6555.288} C_VEL
LIN {X 0,Y 156.541,Z 922.857,A -85,B 0,C 180,E1 6551.375,E2 6551.375} C_VEL
LIN {X 0,Y 161.819,Z 908.772,A -85,B 0,C 180,E1 6548.238,E2 6548.238} C_VEL
LIN {X 0,Y 166.565,Z 893.448,A -85,B 0,C 180,E1 6545.719,E2 6545.719} C_VEL
LIN {X 0,Y 170.45,Z 877.647,A -85,B 0,C 180,E1 6543.805,E2 6543.805} C_VEL
LIN {X 0,Y 173.405,Z 860.617,A -85,B 0,C 180,E1 6542.378,E2 6542.378} C_VEL
LIN {X 0,Y 175.243,Z 843.311,A -85,B 0,C 180,E1 6541.461,E2 6541.461} C_VEL
LIN {X 0,Y 181.141,Z 767.695,A -85,B 0,C 180,E1 6538.877,E2 6538.877} C_VEL
LIN {X 0,Y 179.141,Z 738.152,A -85,B 0,C 180,E1 6536.268,E2 6536.268} C_VEL
LIN {X 0,Y 173.306,Z 725.262,A -85,B 0,C 180,E1 6532.904,E2 6532.904} C_VEL
LIN {X 0,Y 167.648,Z 714.352,A -85,B 0,C 180,E1 6529.239,E2 6529.239} C_VEL
LIN {X 0,Y 163.021,Z 706.607,A -85,B 0,C 180,E1 6525.858,E2 6525.858} C_VEL
LIN {X 0,Y 160.299,Z 701.624,A -85,B 0,C 180,E1 6523.325,E2 6523.325} C_VEL
LIN {X 0,Y 158.744,Z 695.61,A -85,B 0,C 180,E1 6517.66,E2 6517.66} C_VEL
LIN {X 0,Y 157.561,Z 691.066,A -85,B 0,C 180,E1 6512.213,E2 6512.213} C_VEL
LIN {X 0,Y 156.636,Z 687.917,A -85,B 0,C 180,E1 6506.951,E2 6506.951} C_VEL
LIN {X 0,Y 155.966,Z 685.04,A -85,B 0,C 180,E1 6499.085,E2 6499.085} C_VEL
LIN {X 0,Y 155.813,Z 684.743,A -85,B 0,C 180,E1 6492.226,E2 6492.226} C_VEL
LIN {X 0,Y 156.431,Z 685.646,A -85,B 0,C 180,E1 6486.239,E2 6486.239} C_VEL
LIN {X 0,Y 157.876,Z 689.618,A -85,B 0,C 180,E1 6477.823,E2 6477.823} C_VEL
LIN {X 0,Y 159.183,Z 693.439,A -85,B 0,C 180,E1 6472.784,E2 6472.784} C_VEL
LIN {X 0,Y 160.459,Z 697.125,A -85,B 0,C 180,E1 6468.863,E2 6468.863} C_VEL
LIN {X 0,Y 161.486,Z 699.838,A -85,B 0,C 180,E1 6466.575,E2 6466.575} C_VEL
LIN {X 0,Y 166.689,Z 707.629,A -85,B 0,C 180,E1 6462.638,E2 6462.638} C_VEL
LIN {X 0,Y 170.937,Z 714.459,A -85,B 0,C 180,E1 6459.812,E2 6459.812} C_VEL
LIN {X 0,Y 176.266,Z 723.769,A -85,B 0,C 180,E1 6456.65,E2 6456.65} C_VEL
LIN {X 0,Y 182.626,Z 736.312,A -85,B 0,C 180,E1 6453.281,E2 6453.281} C_VEL
LIN {X 0,Y 186.679,Z 745.621,A -85,B 0,C 180,E1 6451.26,E2 6451.26} C_VEL
LIN {X 0,Y 176.977,Z 871.564,A -85,B 0,C 180,E1 6447.257,E2 6447.257} C_VEL
LIN {X 0,Y 174.259,Z 889.781,A -85,B 0,C 180,E1 6446.203,E2 6446.203} C_VEL
LIN {X 0,Y 170.595,Z 906.049,A -85,B 0,C 180,E1 6444.839,E2 6444.839} C_VEL
LIN {X 0,Y 165.704,Z 922.76,A -85,B 0,C 180,E1 6442.887,E2 6442.887} C_VEL
LIN {X 0,Y 160.252,Z 938.15,A -85,B 0,C 180,E1 6440.405,E2 6440.405} C_VEL
LIN {X 0,Y 154.145,Z 953.178,A -85,B 0,C 180,E1 6437.138,E2 6437.138} C_VEL
LIN {X 0,Y 153.558,Z 954.543,A -85,B 0,C 180,E1 6436.793,E2 6436.793} C_VEL
LIN {X 0,Y 150.097,Z 960.404,A -85,B 0,C 180,E1 6435.379,E2 6435.379} C_VEL
LIN {X 0,Y 140.096,Z 971.711,A -85,B 0,C 180,E1 6432.464,E2 6432.464} C_VEL
LIN {X 0,Y 135.571,Z 977.442,A -85,B 0,C 180,E1 6430.348,E2 6430.348} C_VEL
LIN {X 0,Y 134.765,Z 978.865,A -85,B 0,C 180,E1 6429.71,E2 6429.71} C_VEL
LIN {X 0,Y 129.359,Z 989.758,A -85,B 0,C 180,E1 6423.816,E2 6423.816} C_VEL
LIN {X 0,Y 125.196,Z 999.11,A -85,B 0,C 180,E1 6417.08,E2 6417.08} C_VEL
LIN {X 0,Y 122.663,Z 1006.95,A -85,B 0,C 180,E1 6409.525,E2 6409.525} C_VEL
LIN {X 0,Y 122.114,Z 1012.846,A -85,B 0,C 180,E1 6401.813,E2 6401.813} C_VEL
LIN {X 0,Y 123.276,Z 1016.985,A -85,B 0,C 180,E1 6393.964,E2 6393.964} C_VEL
LIN {X 0,Y 124.144,Z 1018.35,A -85,B 0,C 180,E1 6390.001,E2 6390.001} C_VEL
LIN {X 0,Y 122.572,Z 1018.979,A -85,B 0,C 180,E1 6383.913,E2 6383.913} C_VEL
LIN {X 0,Y 121.691,Z 1018.209,A -85,B 0,C 180,E1 6375.245,E2 6375.245} C_VEL
LIN {X 0,Y 123.469,Z 1015.477,A -85,B 0,C 180,E1 6366.216,E2 6366.216} C_VEL
LIN {X 0,Y 128.008,Z 1011.001,A -85,B 0,C 180,E1 6357.918,E2 6357.918} C_VEL
LIN {X 0,Y 135.023,Z 1004.717,A -85,B 0,C 180,E1 6350.444,E2 6350.444} C_VEL
LIN {X 0,Y 143.657,Z 996.895,A -85,B 0,C 180,E1 6344.203,E2 6344.203} C_VEL
LIN {X 0,Y 153.298,Z 987.534,A -85,B 0,C 180,E1 6339.091,E2 6339.091} C_VEL
LIN {X 0,Y 163.442,Z 976.723,A -85,B 0,C 180,E1 6334.941,E2 6334.941} C_VEL
LIN {X 0,Y 173.678,Z 964.422,A -85,B 0,C 180,E1 6331.567,E2 6331.567} C_VEL
LIN {X 0,Y 183.363,Z 951.066,A -85,B 0,C 180,E1 6328.933,E2 6328.933} C_VEL
LIN {X 0,Y 192.031,Z 937.066,A -85,B 0,C 180,E1 6326.935,E2 6326.935} C_VEL
LIN {X 0,Y 200.192,Z 921.295,A -85,B 0,C 180,E1 6325.311,E2 6325.311} C_VEL
LIN {X 0,Y 207.028,Z 904.917,A -85,B 0,C 180,E1 6324.107,E2 6324.107} C_VEL
LIN {X 0,Y 212.414,Z 887.834,A -85,B 0,C 180,E1 6323.21,E2 6323.21} C_VEL
LIN {X 0,Y 216.22,Z 870.079,A -85,B 0,C 180,E1 6322.555,E2 6322.555} C_VEL
LIN {X 0,Y 219.309,Z 843.753,A -85,B 0,C 180,E1 6321.887,E2 6321.887} C_VEL
LIN {X 0,Y 225.799,Z 781.239,A -85,B 0,C 180,E1 6320.408,E2 6320.408} C_VEL
LIN {X 0,Y 223.818,Z 776.941,A -85,B 0,C 180,E1 6318.087,E2 6318.087} C_VEL
LIN {X 0,Y 222.116,Z 773.532,A -85,B 0,C 180,E1 6315.669,E2 6315.669} C_VEL
LIN {X 0,Y 220.415,Z 770.281,A -85,B 0,C 180,E1 6312.576,E2 6312.576} C_VEL
LIN {X 0,Y 219.351,Z 768.49,A -85,B 0,C 180,E1 6309.709,E2 6309.709} C_VEL
LIN {X 0,Y 218.562,Z 767.884,A -85,B 0,C 180,E1 6304.723,E2 6304.723} C_VEL
LIN {X 0,Y 218.702,Z 768.787,A -85,B 0,C 180,E1 6302.358,E2 6302.358} C_VEL
LIN {X 0,Y 219.623,Z 771.323,A -85,B 0,C 180,E1 6298.434,E2 6298.434} C_VEL
LIN {X 0,Y 221.585,Z 776.874,A -85,B 0,C 180,E1 6294.172,E2 6294.172} C_VEL
LIN {X 0,Y 223.561,Z 782.703,A -85,B 0,C 180,E1 6291.123,E2 6291.123} C_VEL
LIN {X 0,Y 224.334,Z 785.241,A -85,B 0,C 180,E1 6290.092,E2 6290.092} C_VEL
LIN {X 0,Y 216.714,Z 854.805,A -85,B 0,C 180,E1 6288.322,E2 6288.322} C_VEL
LIN {X 0,Y 213.587,Z 871.521,A -85,B 0,C 180,E1 6287.558,E2 6287.558} C_VEL
LIN {X 0,Y 208.966,Z 887.937,A -85,B 0,C 180,E1 6286.471,E2 6286.471} C_VEL
LIN {X 0,Y 203.292,Z 902.914,A -85,B 0,C 180,E1 6285.117,E2 6285.117} C_VEL
LIN {X 0,Y 196.206,Z 917.476,A -85,B 0,C 180,E1 6283.343,E2 6283.343} C_VEL
LIN {X 0,Y 188.087,Z 931.063,A -85,B 0,C 180,E1 6281.126,E2 6281.126} C_VEL
LIN {X 0,Y 179.472,Z 942.998,A -85,B 0,C 180,E1 6278.493,E2 6278.493} C_VEL
LIN {X 0,Y 170.509,Z 953.448,A -85,B 0,C 180,E1 6275.355,E2 6275.355} C_VEL
LIN {X 0,Y 161.12,Z 962.794,A -85,B 0,C 180,E1 6271.455,E2 6271.455} C_VEL
LIN {X 0,Y 152.165,Z 970.289,A -85,B 0,C 180,E1 6266.948,E2 6266.948} C_VEL
LIN {X 0,Y 143.389,Z 976.442,A -85,B 0,C 180,E1 6261.35,E2 6261.35} C_VEL
LIN {X 0,Y 136.304,Z 980.458,A -85,B 0,C 180,E1 6255.36,E2 6255.36} C_VEL
LIN {X 0,Y 130.434,Z 982.772,A -85,B 0,C 180,E1 6248.382,E2 6248.382} C_VEL
LIN {X 0,Y 126.461,Z 983.282,A -85,B 0,C 180,E1 6240.925,E2 6240.925} C_VEL
LIN {X 0,Y 124.388,Z 981.979,A -85,B 0,C 180,E1 6233.195,E2 6233.195} C_VEL
LIN {X 0,Y 124.107,Z 978.917,A -85,B 0,C 180,E1 6225.417,E2 6225.417} C_VEL
LIN {X 0,Y 125.395,Z 974.416,A -85,B 0,C 180,E1 6218.251,E2 6218.251} C_VEL
LIN {X 0,Y 128.178,Z 968.118,A -85,B 0,C 180,E1 6211.34,E2 6211.34} C_VEL
LIN {X 0,Y 132.428,Z 959.862,A -85,B 0,C 180,E1 6204.801,E2 6204.801} C_VEL
LIN {X 0,Y 137.319,Z 950.626,A -85,B 0,C 180,E1 6199.418,E2 6199.418} C_VEL
LIN {X 0,Y 142.946,Z 939.494,A -85,B 0,C 180,E1 6194.585,E2 6194.585} C_VEL
LIN {X 0,Y 148.657,Z 927.187,A -85,B 0,C 180,E1 6190.552,E2 6190.552} C_VEL
LIN {X 0,Y 154.075,Z 913.858,A -85,B 0,C 180,E1 6187.286,E2 6187.286} C_VEL
LIN {X 0,Y 159.284,Z 898.833,A -85,B 0,C 180,E1 6184.532,E2 6184.532} C_VEL
LIN {X 0,Y 163.598,Z 883.212,A -85,B 0,C 180,E1 6182.433,E2 6182.433} C_VEL
LIN {X 0,Y 167.129,Z 865.929,A -85,B 0,C 180,E1 6180.793,E2 6180.793} C_VEL
LIN {X 0,Y 169.313,Z 849.145,A -85,B 0,C 180,E1 6179.759,E2 6179.759} C_VEL
LIN {X 0,Y 175.875,Z 768.682,A -85,B 0,C 180,E1 6176.948,E2 6176.948} C_VEL
LIN {X 0,Y 174.325,Z 742.042,A -85,B 0,C 180,E1 6174.535,E2 6174.535} C_VEL
LIN {X 0,Y 169.29,Z 730.513,A -85,B 0,C 180,E1 6171.362,E2 6171.362} C_VEL
LIN {X 0,Y 164.268,Z 720.38,A -85,B 0,C 180,E1 6167.823,E2 6167.823} C_VEL
LIN {X 0,Y 160.081,Z 713.063,A -85,B 0,C 180,E1 6164.539,E2 6164.539} C_VEL
LIN {X 0,Y 156.676,Z 707.336,A -85,B 0,C 180,E1 6161.462,E2 6161.462} C_VEL
LIN {X 0,Y 153.243,Z 701.544,A -85,B 0,C 180,E1 6157.595,E2 6157.595} C_VEL
LIN {X 0,Y 152.133,Z 696.923,A -85,B 0,C 180,E1 6152.022,E2 6152.022} C_VEL
LIN {X 0,Y 151.318,Z 693.862,A -85,B 0,C 180,E1 6146.701,E2 6146.701} C_VEL
LIN {X 0,Y 150.764,Z 691.075,A -85,B 0,C 180,E1 6138.563,E2 6138.563} C_VEL
LIN {X 0,Y 150.717,Z 690.915,A -85,B 0,C 180,E1 6131.48,E2 6131.48} C_VEL
LIN {X 0,Y 151.252,Z 691.719,A -85,B 0,C 180,E1 6126.453,E2 6126.453} C_VEL
LIN {X 0,Y 152.566,Z 695.566,A -85,B 0,C 180,E1 6118.123,E2 6118.123} C_VEL
LIN {X 0,Y 153.725,Z 699.131,A -85,B 0,C 180,E1 6113.277,E2 6113.277} C_VEL
LIN {X 0,Y 155.132,Z 701.537,A -85,B 0,C 180,E1 6111.289,E2 6111.289} C_VEL
LIN {X 0,Y 159.428,Z 707.618,A -85,B 0,C 180,E1 6107.229,E2 6107.229} C_VEL
LIN {X 0,Y 163.75,Z 714.315,A -85,B 0,C 180,E1 6103.779,E2 6103.779} C_VEL
LIN {X 0,Y 168.806,Z 722.707,A -85,B 0,C 180,E1 6100.269,E2 6100.269} C_VEL
LIN {X 0,Y 174.426,Z 733.44,A -85,B 0,C 180,E1 6096.791,E2 6096.791} C_VEL
LIN {X 0,Y 180.343,Z 746.12,A -85,B 0,C 180,E1 6093.538,E2 6093.538} C_VEL
LIN {X 0,Y 181.221,Z 748.485,A -85,B 0,C 180,E1 6093.062,E2 6093.062} C_VEL
LIN {X 0,Y 171.392,Z 870.9,A -85,B 0,C 180,E1 6089.147,E2 6089.147} C_VEL
LIN {X 0,Y 168.595,Z 888.982,A -85,B 0,C 180,E1 6088.096,E2 6088.096} C_VEL
LIN {X 0,Y 164.592,Z 906.069,A -85,B 0,C 180,E1 6086.647,E2 6086.647} C_VEL
LIN {X 0,Y 159.408,Z 922.898,A -85,B 0,C 180,E1 6084.629,E2 6084.629} C_VEL
LIN {X 0,Y 153.532,Z 938.607,A -85,B 0,C 180,E1 6082.001,E2 6082.001} C_VEL
LIN {X 0,Y 147.179,Z 953.415,A -85,B 0,C 180,E1 6078.644,E2 6078.644} C_VEL
LIN {X 0,Y 140.632,Z 967.196,A -85,B 0,C 180,E1 6074.453,E2 6074.453} C_VEL
LIN {X 0,Y 134.765,Z 978.865,A -85,B 0,C 180,E1 6069.71,E2 6069.71} C_VEL
LIN {X 0,Y 131.425,Z 983.616,A -85,B 0,C 180,E1 6067.484,E2 6067.484} C_VEL
LIN {X 0,Y 122.033,Z 992.404,A -85,B 0,C 180,E1 6062.589,E2 6062.589} C_VEL
LIN {X 0,Y 118.235,Z 996.71,A -85,B 0,C 180,E1 6059.34,E2 6059.34} C_VEL
LIN {X 0,Y 117.674,Z 997.753,A -85,B 0,C 180,E1 6058.43,E2 6058.43} C_VEL
LIN {X 0,Y 114.843,Z 1005.651,A -85,B 0,C 180,E1 6050.382,E2 6050.382} C_VEL
LIN {X 0,Y 114.156,Z 1011.586,A -85,B 0,C 180,E1 6042.136,E2 6042.136} C_VEL
LIN {X 0,Y 115.3,Z 1015.674,A -85,B 0,C 180,E1 6033.979,E2 6033.979} C_VEL
LIN {X 0,Y 116.228,Z 1017.022,A -85,B 0,C 180,E1 6030.001,E2 6030.001} C_VEL
LIN {X 0,Y 114.435,Z 1017.691,A -85,B 0,C 180,E1 6022.975,E2 6022.975} C_VEL
LIN {X 0,Y 113.842,Z 1016.913,A -85,B 0,C 180,E1 6013.678,E2 6013.678} C_VEL
LIN {X 0,Y 116.037,Z 1014.348,A -85,B 0,C 180,E1 6004.48,E2 6004.48} C_VEL
LIN {X 0,Y 121.116,Z 1010.017,A -85,B 0,C 180,E1 5995.851,E2 5995.851} C_VEL
LIN {X 0,Y 128.793,Z 1003.831,A -85,B 0,C 180,E1 5988.115,E2 5988.115} C_VEL
LIN {X 0,Y 138.066,Z 996.113,A -85,B 0,C 180,E1 5981.763,E2 5981.763} C_VEL
LIN {X 0,Y 148.285,Z 986.889,A -85,B 0,C 180,E1 5976.641,E2 5976.641} C_VEL
LIN {X 0,Y 158.922,Z 976.189,A -85,B 0,C 180,E1 5972.536,E2 5972.536} C_VEL
LIN {X 0,Y 169.579,Z 964.041,A -85,B 0,C 180,E1 5969.235,E2 5969.235} C_VEL
LIN {X 0,Y 179.602,Z 950.868,A -85,B 0,C 180,E1 5966.682,E2 5966.682} C_VEL
LIN {X 0,Y 188.763,Z 936.676,A -85,B 0,C 180,E1 5964.713,E2 5964.713} C_VEL
LIN {X 0,Y 196.904,Z 921.516,A -85,B 0,C 180,E1 5963.206,E2 5963.206} C_VEL
LIN {X 0,Y 203.897,Z 905.412,A -85,B 0,C 180,E1 5962.058,E2 5962.058} C_VEL
LIN {X 0,Y 209.626,Z 888.141,A -85,B 0,C 180,E1 5961.176,E2 5961.176} C_VEL
LIN {X 0,Y 213.614,Z 870.41,A -85,B 0,C 180,E1 5960.54,E2 5960.54} C_VEL
LIN {X 0,Y 216.673,Z 845.921,A -85,B 0,C 180,E1 5959.929,E2 5959.929} C_VEL
LIN {X 0,Y 223.06,Z 786.22,A -85,B 0,C 180,E1 5958.557,E2 5958.557} C_VEL
LIN {X 0,Y 220.831,Z 781.359,A -85,B 0,C 180,E1 5955.335,E2 5955.335} C_VEL
LIN {X 0,Y 219.159,Z 777.981,A -85,B 0,C 180,E1 5952.114,E2 5952.114} C_VEL
LIN {X 0,Y 218.262,Z 776.378,A -85,B 0,C 180,E1 5949.492,E2 5949.492} C_VEL
LIN {X 0,Y 217.545,Z 775.852,A -85,B 0,C 180,E1 5944.481,E2 5944.481} C_VEL
LIN {X 0,Y 218.368,Z 778.862,A -85,B 0,C 180,E1 5939.081,E2 5939.081} C_VEL
LIN {X 0,Y 220.088,Z 784.304,A -85,B 0,C 180,E1 5934.852,E2 5934.852} C_VEL
LIN {X 0,Y 221.78,Z 789.767,A -85,B 0,C 180,E1 5931.978,E2 5931.978} C_VEL
LIN {X 0,Y 214.309,Z 855.759,A -85,B 0,C 180,E1 5930.336,E2 5930.336} C_VEL
LIN {X 0,Y 211.037,Z 872.505,A -85,B 0,C 180,E1 5929.587,E2 5929.587} C_VEL
LIN {X 0,Y 206.109,Z 889.337,A -85,B 0,C 180,E1 5928.499,E2 5928.499} C_VEL
LIN {X 0,Y 199.995,Z 904.719,A -85,B 0,C 180,E1 5927.131,E2 5927.131} C_VEL
LIN {X 0,Y 192.69,Z 919.108,A -85,B 0,C 180,E1 5925.406,E2 5925.406} C_VEL
LIN {X 0,Y 184.547,Z 932.201,A -85,B 0,C 180,E1 5923.312,E2 5923.312} C_VEL
LIN {X 0,Y 175.473,Z 944.261,A -85,B 0,C 180,E1 5920.701,E2 5920.701} C_VEL
LIN {X 0,Y 165.652,Z 955.173,A -85,B 0,C 180,E1 5917.441,E2 5917.441} C_VEL
LIN {X 0,Y 156.157,Z 964.119,A -85,B 0,C 180,E1 5913.689,E2 5913.689} C_VEL
LIN {X 0,Y 146.711,Z 971.564,A -85,B 0,C 180,E1 5909.171,E2 5909.171} C_VEL
LIN {X 0,Y 137.686,Z 977.491,A -85,B 0,C 180,E1 5903.712,E2 5903.712} C_VEL
LIN {X 0,Y 130.01,Z 981.561,A -85,B 0,C 180,E1 5897.586,E2 5897.586} C_VEL
LIN {X 0,Y 123.543,Z 983.943,A -85,B 0,C 180,E1 5890.349,E2 5890.349} C_VEL
LIN {X 0,Y 119.056,Z 984.512,A -85,B 0,C 180,E1 5882.512,E2 5882.512} C_VEL
LIN {X 0,Y 116.618,Z 983.304,A -85,B 0,C 180,E1 5874.301,E2 5874.301} C_VEL
LIN {X 0,Y 116.132,Z 980.306,A -85,B 0,C 180,E1 5865.991,E2 5865.991} C_VEL
LIN {X 0,Y 117.511,Z 975.542,A -85,B 0,C 180,E1 5857.824,E2 5857.824} C_VEL
LIN {X 0,Y 120.467,Z 969.227,A -85,B 0,C 180,E1 5850.475,E2 5850.475} C_VEL
LIN {X 0,Y 124.99,Z 960.962,A -85,B 0,C 180,E1 5843.569,E2 5843.569} C_VEL
LIN {X 0,Y 130.085,Z 951.908,A -85,B 0,C 180,E1 5838.022,E2 5838.022} C_VEL
LIN {X 0,Y 136.13,Z 940.613,A -85,B 0,C 180,E1 5832.914,E2 5832.914} C_VEL
LIN {X 0,Y 142.148,Z 928.33,A -85,B 0,C 180,E1 5828.761,E2 5828.761} C_VEL
LIN {X 0,Y 147.839,Z 915.067,A -85,B 0,C 180,E1 5825.421,E2 5825.421} C_VEL
LIN {X 0,Y 153.292,Z 900.117,A -85,B 0,C 180,E1 5822.622,E2 5822.622} C_VEL
LIN {X 0,Y 157.781,Z 884.793,A -85,B 0,C 180,E1 5820.51,E2 5820.51} C_VEL
LIN {X 0,Y 161.496,Z 867.652,A -85,B 0,C 180,E1 5818.844,E2 5818.844} C_VEL
LIN {X 0,Y 163.891,Z 850.773,A -85,B 0,C 180,E1 5817.761,E2 5817.761} C_VEL
LIN {X 0,Y 170.793,Z 769.706,A -85,B 0,C 180,E1 5814.914,E2 5814.914} C_VEL
LIN {X 0,Y 169.592,Z 745.653,A -85,B 0,C 180,E1 5812.645,E2 5812.645} C_VEL
LIN {X 0,Y 164.873,Z 734.621,A -85,B 0,C 180,E1 5809.361,E2 5809.361} C_VEL
LIN {X 0,Y 160.409,Z 725.396,A -85,B 0,C 180,E1 5805.922,E2 5805.922} C_VEL
LIN {X 0,Y 157.095,Z 719.282,A -85,B 0,C 180,E1 5803.049,E2 5803.049} C_VEL
LIN {X 0,Y 154.19,Z 714.12,A -85,B 0,C 180,E1 5800.183,E2 5800.183} C_VEL
LIN {X 0,Y 150.573,Z 708.08,A -85,B 0,C 180,E1 5795.97,E2 5795.97} C_VEL
LIN {X 0,Y 146.747,Z 702.161,A -85,B 0,C 180,E1 5790.079,E2 5790.079} C_VEL
LIN {X 0,Y 145.971,Z 699.727,A -85,B 0,C 180,E1 5786.191,E2 5786.191} C_VEL
LIN {X 0,Y 145.589,Z 697.168,A -85,B 0,C 180,E1 5778.417,E2 5778.417} C_VEL
LIN {X 0,Y 145.61,Z 697.077,A -85,B 0,C 180,E1 5771.086,E2 5771.086} C_VEL
LIN {X 0,Y 146.091,Z 697.947,A -85,B 0,C 180,E1 5766.288,E2 5766.288} C_VEL
LIN {X 0,Y 147.041,Z 700.577,A -85,B 0,C 180,E1 5760.605,E2 5760.605} C_VEL
LIN {X 0,Y 148.873,Z 703.232,A -85,B 0,C 180,E1 5757.499,E2 5757.499} C_VEL
LIN {X 0,Y 152.131,Z 707.451,A -85,B 0,C 180,E1 5753.311,E2 5753.311} C_VEL
LIN {X 0,Y 156.769,Z 714.292,A -85,B 0,C 180,E1 5748.504,E2 5748.504} C_VEL
LIN {X 0,Y 160.983,Z 721.175,A -85,B 0,C 180,E1 5744.88,E2 5744.88} C_VEL
LIN {X 0,Y 165.986,Z 729.897,A -85,B 0,C 180,E1 5741.2,E2 5741.2} C_VEL
LIN {X 0,Y 172.018,Z 742.175,A -85,B 0,C 180,E1 5737.262,E2 5737.262} C_VEL
LIN {X 0,Y 175.904,Z 751.331,A -85,B 0,C 180,E1 5734.96,E2 5734.96} C_VEL
LIN {X 0,Y 165.943,Z 870.389,A -85,B 0,C 180,E1 5731.141,E2 5731.141} C_VEL
LIN {X 0,Y 163.015,Z 888.574,A -85,B 0,C 180,E1 5730.078,E2 5730.078} C_VEL
LIN {X 0,Y 158.754,Z 906.024,A -85,B 0,C 180,E1 5728.586,E2 5728.586} C_VEL
LIN {X 0,Y 153.382,Z 922.648,A -85,B 0,C 180,E1 5726.555,E2 5726.555} C_VEL
LIN {X 0,Y 147.269,Z 938.262,A -85,B 0,C 180,E1 5723.896,E2 5723.896} C_VEL
LIN {X 0,Y 140.642,Z 952.977,A -85,B 0,C 180,E1 5720.477,E2 5720.477} C_VEL
LIN {X 0,Y 133.767,Z 966.672,A -85,B 0,C 180,E1 5716.164,E2 5716.164} C_VEL
LIN {X 0,Y 127.08,Z 979.153,A -85,B 0,C 180,E1 5710.772,E2 5710.772} C_VEL
LIN {X 0,Y 121.159,Z 990.418,A -85,B 0,C 180,E1 5704.138,E2 5704.138} C_VEL
LIN {X 0,Y 117.674,Z 997.753,A -85,B 0,C 180,E1 5698.43,E2 5698.43} C_VEL
LIN {X 0,Y 115.272,Z 1001.197,A -85,B 0,C 180,E1 5695.213,E2 5695.213} C_VEL
LIN {X 0,Y 109.379,Z 1006.175,A -85,B 0,C 180,E1 5689.248,E2 5689.248} C_VEL
LIN {X 0,Y 106.472,Z 1009.238,A -85,B 0,C 180,E1 5684.394,E2 5684.394} C_VEL
LIN {X 0,Y 106.204,Z 1010.388,A -85,B 0,C 180,E1 5682.39,E2 5682.39} C_VEL
LIN {X 0,Y 107.378,Z 1014.446,A -85,B 0,C 180,E1 5673.738,E2 5673.738} C_VEL
LIN {X 0,Y 108.183,Z 1015.772,A -85,B 0,C 180,E1 5669.471,E2 5669.471} C_VEL
LIN {X 0,Y 106.138,Z 1016.424,A -85,B 0,C 180,E1 5660.786,E2 5660.786} C_VEL
LIN {X 0,Y 106.239,Z 1015.406,A -85,B 0,C 180,E1 5650.769,E2 5650.769} C_VEL
LIN {X 0,Y 109.699,Z 1012.447,A -85,B 0,C 180,E1 5640.516,E2 5640.516} C_VEL
LIN {X 0,Y 116.121,Z 1007.797,A -85,B 0,C 180,E1 5631.586,E2 5631.586} C_VEL
LIN {X 0,Y 124.979,Z 1001.36,A -85,B 0,C 180,E1 5623.945,E2 5623.945} C_VEL
LIN {X 0,Y 135.332,Z 993.228,A -85,B 0,C 180,E1 5617.765,E2 5617.765} C_VEL
LIN {X 0,Y 146.449,Z 983.626,A -85,B 0,C 180,E1 5612.886,E2 5612.886} C_VEL
LIN {X 0,Y 157.805,Z 972.535,A -85,B 0,C 180,E1 5609.03,E2 5609.03} C_VEL
LIN {X 0,Y 168.635,Z 960.308,A -85,B 0,C 180,E1 5606.07,E2 5606.07} C_VEL
LIN {X 0,Y 179.098,Z 946.466,A -85,B 0,C 180,E1 5603.714,E2 5603.714} C_VEL
LIN {X 0,Y 188.601,Z 931.521,A -85,B 0,C 180,E1 5601.914,E2 5601.914} C_VEL
LIN {X 0,Y 196.559,Z 916.31,A -85,B 0,C 180,E1 5600.615,E2 5600.615} C_VEL
LIN {X 0,Y 203.283,Z 900.022,A -85,B 0,C 180,E1 5599.627,E2 5599.627} C_VEL
LIN {X 0,Y 208.791,Z 882.088,A -85,B 0,C 180,E1 5598.848,E2 5598.848} C_VEL
LIN {X 0,Y 212.4,Z 864.329,A -85,B 0,C 180,E1 5598.3,E2 5598.3} C_VEL
LIN {X 0,Y 220.572,Z 791.596,A -85,B 0,C 180,E1 5596.654,E2 5596.654} C_VEL
LIN {X 0,Y 218.999,Z 788.049,A -85,B 0,C 180,E1 5594.003,E2 5594.003} C_VEL
LIN {X 0,Y 217.647,Z 785.087,A -85,B 0,C 180,E1 5590.856,E2 5590.856} C_VEL
LIN {X 0,Y 216.862,Z 783.957,A -85,B 0,C 180,E1 5587.95,E2 5587.95} C_VEL
LIN {X 0,Y 216.537,Z 783.918,A -85,B 0,C 180,E1 5583.971,E2 5583.971} C_VEL
LIN {X 0,Y 217.274,Z 786.895,A -85,B 0,C 180,E1 5579.208,E2 5579.208} C_VEL
LIN {X 0,Y 218.682,Z 791.958,A -85,B 0,C 180,E1 5575.41,E2 5575.41} C_VEL
LIN {X 0,Y 219.439,Z 794.812,A -85,B 0,C 180,E1 5573.895,E2 5573.895} C_VEL
LIN {X 0,Y 212.24,Z 856.613,A -85,B 0,C 180,E1 5572.399,E2 5572.399} C_VEL
LIN {X 0,Y 208.83,Z 873.463,A -85,B 0,C 180,E1 5571.669,E2 5571.669} C_VEL
LIN {X 0,Y 204.105,Z 889.226,A -85,B 0,C 180,E1 5570.696,E2 5570.696} C_VEL
LIN {X 0,Y 197.853,Z 904.762,A -85,B 0,C 180,E1 5569.392,E2 5569.392} C_VEL
LIN {X 0,Y 190.313,Z 919.277,A -85,B 0,C 180,E1 5567.741,E2 5567.741} C_VEL
LIN {X 0,Y 181.567,Z 932.935,A -85,B 0,C 180,E1 5565.652,E2 5565.652} C_VEL
LIN {X 0,Y 172.118,Z 945.101,A -85,B 0,C 180,E1 5563.114,E2 5563.114} C_VEL
LIN {X 0,Y 161.814,Z 956.116,A -85,B 0,C 180,E1 5559.92,E2 5559.92} C_VEL
LIN {X 0,Y 151.857,Z 965.091,A -85,B 0,C 180,E1 5556.234,E2 5556.234} C_VEL
LIN {X 0,Y 141.877,Z 972.59,A -85,B 0,C 180,E1 5551.752,E2 5551.752} C_VEL
LIN {X 0,Y 132.242,Z 978.557,A -85,B 0,C 180,E1 5546.272,E2 5546.272} C_VEL
LIN {X 0,Y 123.936,Z 982.67,A -85,B 0,C 180,E1 5540.032,E2 5540.032} C_VEL
LIN {X 0,Y 116.817,Z 985.119,A -85,B 0,C 180,E1 5532.545,E2 5532.545} C_VEL
LIN {X 0,Y 111.513,Z 985.733,A -85,B 0,C 180,E1 5523.772,E2 5523.772} C_VEL
LIN {X 0,Y 108.786,Z 984.481,A -85,B 0,C 180,E1 5515.01,E2 5515.01} C_VEL
LIN {X 0,Y 108.194,Z 981.424,A -85,B 0,C 180,E1 5506.028,E2 5506.028} C_VEL
LIN {X 0,Y 109.632,Z 976.667,A -85,B 0,C 180,E1 5497.335,E2 5497.335} C_VEL
LIN {X 0,Y 112.788,Z 970.335,A -85,B 0,C 180,E1 5489.491,E2 5489.491} C_VEL
LIN {X 0,Y 117.616,Z 962.062,A -85,B 0,C 180,E1 5482.182,E2 5482.182} C_VEL
LIN {X 0,Y 123.037,Z 953.013,A -85,B 0,C 180,E1 5476.368,E2 5476.368} C_VEL
LIN {X 0,Y 129.442,Z 941.731,A -85,B 0,C 180,E1 5471.068,E2 5471.068} C_VEL
LIN {X 0,Y 136.082,Z 928.891,A -85,B 0,C 180,E1 5466.623,E2 5466.623} C_VEL
LIN {X 0,Y 142.081,Z 915.524,A -85,B 0,C 180,E1 5463.231,E2 5463.231} C_VEL
LIN {X 0,Y 147.809,Z 900.482,A -85,B 0,C 180,E1 5460.407,E2 5460.407} C_VEL
LIN {X 0,Y 152.392,Z 885.448,A -85,B 0,C 180,E1 5458.338,E2 5458.338} C_VEL
LIN {X 0,Y 156.292,Z 868.196,A -85,B 0,C 180,E1 5456.661,E2 5456.661} C_VEL
LIN {X 0,Y 158.79,Z 851.296,A -85,B 0,C 180,E1 5455.579,E2 5455.579} C_VEL
LIN {X 0,Y 165.937,Z 770.658,A -85,B 0,C 180,E1 5452.751,E2 5452.751} C_VEL
LIN {X 0,Y 165.095,Z 749.494,A -85,B 0,C 180,E1 5450.687,E2 5450.687} C_VEL
LIN {X 0,Y 160.26,Z 737.718,A -85,B 0,C 180,E1 5446.95,E2 5446.95} C_VEL
LIN {X 0,Y 155.573,Z 727.897,A -85,B 0,C 180,E1 5442.817,E2 5442.817} C_VEL
LIN {X 0,Y 151.784,Z 720.903,A -85,B 0,C 180,E1 5438.863,E2 5438.863} C_VEL
LIN {X 0,Y 148.561,Z 715.217,A -85,B 0,C 180,E1 5434.804,E2 5434.804} C_VEL
LIN {X 0,Y 144.949,Z 709.223,A -85,B 0,C 180,E1 5428.648,E2 5428.648} C_VEL
LIN {X 0,Y 143.522,Z 707.072,A -85,B 0,C 180,E1 5425.149,E2 5425.149} C_VEL
LIN {X 0,Y 142.019,Z 704.301,A -85,B 0,C 180,E1 5418.047,E2 5418.047} C_VEL
LIN {X 0,Y 142.357,Z 704.418,A -85,B 0,C 180,E1 5410.478,E2 5410.478} C_VEL
LIN {X 0,Y 143.466,Z 705.626,A -85,B 0,C 180,E1 5406.202,E2 5406.202} C_VEL
LIN {X 0,Y 146.385,Z 709.318,A -85,B 0,C 180,E1 5399.805,E2 5399.805} C_VEL
LIN {X 0,Y 150.184,Z 714.802,A -85,B 0,C 180,E1 5394.269,E2 5394.269} C_VEL
LIN {X 0,Y 154.448,Z 721.431,A -85,B 0,C 180,E1 5389.557,E2 5389.557} C_VEL
LIN {X 0,Y 158.677,Z 728.712,A -85,B 0,C 180,E1 5385.682,E2 5385.682} C_VEL
LIN {X 0,Y 163.889,Z 738.565,A -85,B 0,C 180,E1 5381.643,E2 5381.643} C_VEL
LIN {X 0,Y 169.428,Z 750.684,A -85,B 0,C 180,E1 5377.856,E2 5377.856} C_VEL
LIN {X 0,Y 170.779,Z 754.306,A -85,B 0,C 180,E1 5376.97,E2 5376.97} C_VEL
LIN {X 0,Y 160.717,Z 869.687,A -85,B 0,C 180,E1 5373.273,E2 5373.273} C_VEL
LIN {X 0,Y 157.694,Z 887.811,A -85,B 0,C 180,E1 5372.217,E2 5372.217} C_VEL
LIN {X 0,Y 153.489,Z 904.54,A -85,B 0,C 180,E1 5370.8,E2 5370.8} C_VEL
LIN {X 0,Y 148.274,Z 920.392,A -85,B 0,C 180,E1 5368.917,E2 5368.917} C_VEL
LIN {X 0,Y 141.871,Z 936.277,A -85,B 0,C 180,E1 5366.268,E2 5366.268} C_VEL
LIN {X 0,Y 134.891,Z 951.169,A -85,B 0,C 180,E1 5362.83,E2 5362.83} C_VEL
LIN {X 0,Y 127.607,Z 965.034,A -85,B 0,C 180,E1 5358.444,E2 5358.444} C_VEL
LIN {X 0,Y 120.906,Z 976.893,A -85,B 0,C 180,E1 5353.304,E2 5353.304} C_VEL
LIN {X 0,Y 114.799,Z 987.646,A -85,B 0,C 180,E1 5346.94,E2 5346.94} C_VEL
LIN {X 0,Y 109.861,Z 997.165,A -85,B 0,C 180,E1 5339.245,E2 5339.245} C_VEL
LIN {X 0,Y 106.912,Z 1004.856,A -85,B 0,C 180,E1 5330.739,E2 5330.739} C_VEL
LIN {X 0,Y 106.204,Z 1010.388,A -85,B 0,C 180,E1 5322.39,E2 5322.39} C_VEL
LIN {X 0,Y 105.501,Z 1011.88,A -85,B 0,C 180,E1 5319.304,E2 5319.304} C_VEL
LIN {X 0,Y 102.782,Z 1013.363,A -85,B 0,C 180,E1 5314.614,E2 5314.614} C_VEL
LIN {X 0,Y 100.27,Z 1014.358,A -85,B 0,C 180,E1 5309.642,E2 5309.642} C_VEL
LIN {X 0,Y 98.133,Z 1015.114,A -85,B 0,C 180,E1 5300.027,E2 5300.027} C_VEL
LIN {X 0,Y 98.598,Z 1014.175,A -85,B 0,C 180,E1 5288.896,E2 5288.896} C_VEL
LIN {X 0,Y 102.624,Z 1011.371,A -85,B 0,C 180,E1 5278.257,E2 5278.257} C_VEL
LIN {X 0,Y 110.194,Z 1006.566,A -85,B 0,C 180,E1 5268.52,E2 5268.52} C_VEL
LIN {X 0,Y 120.032,Z 1000.094,A -85,B 0,C 180,E1 5260.711,E2 5260.711} C_VEL
LIN {X 0,Y 131.177,Z 991.983,A -85,B 0,C 180,E1 5254.595,E2 5254.595} C_VEL
LIN {X 0,Y 142.955,Z 982.372,A -85,B 0,C 180,E1 5249.857,E2 5249.857} C_VEL
LIN {X 0,Y 154.842,Z 971.261,A -85,B 0,C 180,E1 5246.161,E2 5246.161} C_VEL
LIN {X 0,Y 166.091,Z 958.985,A -85,B 0,C 180,E1 5243.359,E2 5243.359} C_VEL
LIN {X 0,Y 176.452,Z 945.698,A -85,B 0,C 180,E1 5241.231,E2 5241.231} C_VEL
LIN {X 0,Y 186.186,Z 930.864,A -85,B 0,C 180,E1 5239.549,E2 5239.549} C_VEL
LIN {X 0,Y 194.344,Z 915.734,A -85,B 0,C 180,E1 5238.34,E2 5238.34} C_VEL
LIN {X 0,Y 201.205,Z 899.597,A -85,B 0,C 180,E1 5237.425,E2 5237.425} C_VEL
LIN {X 0,Y 206.757,Z 882.065,A -85,B 0,C 180,E1 5236.71,E2 5236.71} C_VEL
LIN {X 0,Y 210.536,Z 864.233,A -85,B 0,C 180,E1 5236.187,E2 5236.187} C_VEL
LIN {X 0,Y 218.327,Z 797.085,A -85,B 0,C 180,E1 5234.724,E2 5234.724} C_VEL
LIN {X 0,Y 216.711,Z 793.385,A -85,B 0,C 180,E1 5231.173,E2 5231.173} C_VEL
LIN {X 0,Y 216.026,Z 792.086,A -85,B 0,C 180,E1 5228.785,E2 5228.785} C_VEL
LIN {X 0,Y 215.505,Z 791.779,A -85,B 0,C 180,E1 5224.257,E2 5224.257} C_VEL
LIN {X 0,Y 216.084,Z 794.552,A -85,B 0,C 180,E1 5219.734,E2 5219.734} C_VEL
LIN {X 0,Y 217.215,Z 799.271,A -85,B 0,C 180,E1 5216.172,E2 5216.172} C_VEL
LIN {X 0,Y 217.318,Z 800.087,A -85,B 0,C 180,E1 5215.846,E2 5215.846} C_VEL
LIN {X 0,Y 210.462,Z 857.392,A -85,B 0,C 180,E1 5214.504,E2 5214.504} C_VEL
LIN {X 0,Y 206.931,Z 874.318,A -85,B 0,C 180,E1 5213.799,E2 5213.799} C_VEL
LIN {X 0,Y 201.806,Z 890.838,A -85,B 0,C 180,E1 5212.816,E2 5212.816} C_VEL
LIN {X 0,Y 195.566,Z 905.782,A -85,B 0,C 180,E1 5211.607,E2 5211.607} C_VEL
LIN {X 0,Y 187.809,Z 920.274,A -85,B 0,C 180,E1 5210.031,E2 5210.031} C_VEL
LIN {X 0,Y 178.853,Z 933.835,A -85,B 0,C 180,E1 5208.046,E2 5208.046} C_VEL
LIN {X 0,Y 169.111,Z 945.964,A -85,B 0,C 180,E1 5205.621,E2 5205.621} C_VEL
LIN {X 0,Y 159.121,Z 956.301,A -85,B 0,C 180,E1 5202.767,E2 5202.767} C_VEL
LIN {X 0,Y 147.875,Z 966.064,A -85,B 0,C 180,E1 5198.92,E2 5198.92} C_VEL
LIN {X 0,Y 137.353,Z 973.616,A -85,B 0,C 180,E1 5194.508,E2 5194.508} C_VEL
LIN {X 0,Y 127.084,Z 979.62,A -85,B 0,C 180,E1 5189.045,E2 5189.045} C_VEL
LIN {X 0,Y 117.568,Z 984.009,A -85,B 0,C 180,E1 5182.271,E2 5182.271} C_VEL
LIN {X 0,Y 109.862,Z 986.386,A -85,B 0,C 180,E1 5174.488,E2 5174.488} C_VEL
LIN {X 0,Y 104.036,Z 986.955,A -85,B 0,C 180,E1 5165.221,E2 5165.221} C_VEL
LIN {X 0,Y 100.971,Z 985.651,A -85,B 0,C 180,E1 5155.829,E2 5155.829} C_VEL
LIN {X 0,Y 100.248,Z 982.596,A -85,B 0,C 180,E1 5146.216,E2 5146.216} C_VEL
LIN {X 0,Y 101.762,Z 977.788,A -85,B 0,C 180,E1 5136.77,E2 5136.77} C_VEL
LIN {X 0,Y 105.146,Z 971.441,A -85,B 0,C 180,E1 5128.364,E2 5128.364} C_VEL
LIN {X 0,Y 110.321,Z 963.162,A -85,B 0,C 180,E1 5120.61,E2 5120.61} C_VEL
LIN {X 0,Y 116.313,Z 953.774,A -85,B 0,C 180,E1 5114.324,E2 5114.324} C_VEL
LIN {X 0,Y 122.903,Z 942.849,A -85,B 0,C 180,E1 5109.024,E2 5109.024} C_VEL
LIN {X 0,Y 129.916,Z 930.038,A -85,B 0,C 180,E1 5104.469,E2 5104.469} C_VEL
LIN {X 0,Y 136.223,Z 916.734,A -85,B 0,C 180,E1 5101.024,E2 5101.024} C_VEL
LIN {X 0,Y 142.222,Z 901.765,A -85,B 0,C 180,E1 5098.178,E2 5098.178} C_VEL
LIN {X 0,Y 147.017,Z 886.923,A -85,B 0,C 180,E1 5096.103,E2 5096.103} C_VEL
LIN {X 0,Y 151.092,Z 869.918,A -85,B 0,C 180,E1 5094.427,E2 5094.427} C_VEL
LIN {X 0,Y 153.85,Z 852.638,A -85,B 0,C 180,E1 5093.294,E2 5093.294} C_VEL
LIN {X 0,Y 161.333,Z 771.698,A -85,B 0,C 180,E1 5090.47,E2 5090.47} C_VEL
LIN {X 0,Y 160.762,Z 753.306,A -85,B 0,C 180,E1 5088.611,E2 5088.611} C_VEL
LIN {X 0,Y 156.656,Z 742.92,A -85,B 0,C 180,E1 5085.111,E2 5085.111} C_VEL
LIN {X 0,Y 152.618,Z 733.978,A -85,B 0,C 180,E1 5081.155,E2 5081.155} C_VEL
LIN {X 0,Y 149.442,Z 727.684,A -85,B 0,C 180,E1 5077.507,E2 5077.507} C_VEL
LIN {X 0,Y 146.571,Z 722.284,A -85,B 0,C 180,E1 5073.543,E2 5073.543} C_VEL
LIN {X 0,Y 143.36,Z 716.498,A -85,B 0,C 180,E1 5067.408,E2 5067.408} C_VEL
LIN {X 0,Y 142.01,Z 714.459,A -85,B 0,C 180,E1 5063.662,E2 5063.662} C_VEL
LIN {X 0,Y 140.995,Z 712.213,A -85,B 0,C 180,E1 5057.755,E2 5057.755} C_VEL
LIN {X 0,Y 141.409,Z 712.413,A -85,B 0,C 180,E1 5050.182,E2 5050.182} C_VEL
LIN {X 0,Y 142.425,Z 713.669,A -85,B 0,C 180,E1 5046.248,E2 5046.248} C_VEL
LIN {X 0,Y 144.883,Z 716.944,A -85,B 0,C 180,E1 5040.594,E2 5040.594} C_VEL
LIN {X 0,Y 148.343,Z 722.261,A -85,B 0,C 180,E1 5035.168,E2 5035.168} C_VEL
LIN {X 0,Y 152.182,Z 728.562,A -85,B 0,C 180,E1 5030.642,E2 5030.642} C_VEL
LIN {X 0,Y 156.304,Z 736.089,A -85,B 0,C 180,E1 5026.593,E2 5026.593} C_VEL
LIN {X 0,Y 161.044,Z 745.701,A -85,B 0,C 180,E1 5022.662,E2 5022.662} C_VEL
LIN {X 0,Y 165.889,Z 757.111,A -85,B 0,C 180,E1 5019.107,E2 5019.107} C_VEL
LIN {X 0,Y 155.71,Z 869.108,A -85,B 0,C 180,E1 5015.538,E2 5015.538} C_VEL
LIN {X 0,Y 152.552,Z 887.305,A -85,B 0,C 180,E1 5014.482,E2 5014.482} C_VEL
LIN {X 0,Y 148.079,Z 904.394,A -85,B 0,C 180,E1 5013.038,E2 5013.038} C_VEL
LIN {X 0,Y 142.674,Z 920.08,A -85,B 0,C 180,E1 5011.166,E2 5011.166} C_VEL
LIN {X 0,Y 136.013,Z 935.84,A -85,B 0,C 180,E1 5008.513,E2 5008.513} C_VEL
LIN {X 0,Y 128.716,Z 950.648,A -85,B 0,C 180,E1 5005.038,E2 5005.038} C_VEL
LIN {X 0,Y 121.366,Z 963.902,A -85,B 0,C 180,E1 5000.753,E2 5000.753} C_VEL
LIN {X 0,Y 114.007,Z 976.144,A -85,B 0,C 180,E1 4995.268,E2 4995.268} C_VEL
LIN {X 0,Y 107.467,Z 986.887,A -85,B 0,C 180,E1 4988.564,E2 4988.564} C_VEL
LIN {X 0,Y 102.263,Z 996.166,A -85,B 0,C 180,E1 4980.56,E2 4980.56} C_VEL
LIN {X 0,Y 99.021,Z 1003.919,A -85,B 0,C 180,E1 4971.317,E2 4971.317} C_VEL
LIN {X 0,Y 98.287,Z 1009.665,A -85,B 0,C 180,E1 4961.74,E2 4961.74} C_VEL
LIN {X 0,Y 99.734,Z 1013.578,A -85,B 0,C 180,E1 4952.299,E2 4952.299} C_VEL
LIN {X 0,Y 100.27,Z 1014.358,A -85,B 0,C 180,E1 4949.642,E2 4949.642} C_VEL
LIN {X 0,Y 98.319,Z 1014.826,A -85,B 0,C 180,E1 4945.655,E2 4945.655} C_VEL
LIN {X 0,Y 94.002,Z 1014.572,A -85,B 0,C 180,E1 4939.502,E2 4939.502} C_VEL
LIN {X 0,Y 90.611,Z 1013.627,A -85,B 0,C 180,E1 4932.114,E2 4932.114} C_VEL
LIN {X 0,Y 90.608,Z 1013.204,A -85,B 0,C 180,E1 4928.934,E2 4928.934} C_VEL
LIN {X 0,Y 94.711,Z 1010.852,A -85,B 0,C 180,E1 4917.426,E2 4917.426} C_VEL
LIN {X 0,Y 102.13,Z 1006.787,A -85,B 0,C 180,E1 4907.507,E2 4907.507} C_VEL
LIN {X 0,Y 112.333,Z 1000.788,A -85,B 0,C 180,E1 4899.194,E2 4899.194} C_VEL
LIN {X 0,Y 124.367,Z 992.927,A -85,B 0,C 180,E1 4892.591,E2 4892.591} C_VEL
LIN {X 0,Y 136.689,Z 983.765,A -85,B 0,C 180,E1 4887.738,E2 4887.738} C_VEL
LIN {X 0,Y 148.917,Z 973.165,A -85,B 0,C 180,E1 4884.06,E2 4884.06} C_VEL
LIN {X 0,Y 160.873,Z 961.1,A -85,B 0,C 180,E1 4881.208,E2 4881.208} C_VEL
LIN {X 0,Y 171.91,Z 948.013,A -85,B 0,C 180,E1 4879.069,E2 4879.069} C_VEL
LIN {X 0,Y 181.853,Z 933.914,A -85,B 0,C 180,E1 4877.46,E2 4877.46} C_VEL
LIN {X 0,Y 190.589,Z 918.802,A -85,B 0,C 180,E1 4876.252,E2 4876.252} C_VEL
LIN {X 0,Y 198.031,Z 902.722,A -85,B 0,C 180,E1 4875.343,E2 4875.343} C_VEL
LIN {X 0,Y 203.866,Z 886.203,A -85,B 0,C 180,E1 4874.669,E2 4874.669} C_VEL
LIN {X 0,Y 208.13,Z 868.623,A -85,B 0,C 180,E1 4874.15,E2 4874.15} C_VEL
LIN {X 0,Y 211.425,Z 844.606,A -85,B 0,C 180,E1 4873.628,E2 4873.628} C_VEL
LIN {X 0,Y 216.262,Z 803.074,A -85,B 0,C 180,E1 4872.741,E2 4872.741} C_VEL
LIN {X 0,Y 215.151,Z 800.203,A -85,B 0,C 180,E1 4869.36,E2 4869.36} C_VEL
LIN {X 0,Y 214.474,Z 799.666,A -85,B 0,C 180,E1 4864.545,E2 4864.545} C_VEL
LIN {X 0,Y 214.931,Z 802.393,A -85,B 0,C 180,E1 4860.133,E2 4860.133} C_VEL
LIN {X 0,Y 215.472,Z 805.375,A -85,B 0,C 180,E1 4857.834,E2 4857.834} C_VEL
LIN {X 0,Y 208.934,Z 858.398,A -85,B 0,C 180,E1 4856.633,E2 4856.633} C_VEL
LIN {X 0,Y 205.263,Z 875.398,A -85,B 0,C 180,E1 4855.953,E2 4855.953} C_VEL
LIN {X 0,Y 200.001,Z 891.861,A -85,B 0,C 180,E1 4855.02,E2 4855.02} C_VEL
LIN {X 0,Y 193.578,Z 906.801,A -85,B 0,C 180,E1 4853.872,E2 4853.872} C_VEL
LIN {X 0,Y 185.613,Z 921.271,A -85,B 0,C 180,E1 4852.379,E2 4852.379} C_VEL
LIN {X 0,Y 176.396,Z 934.822,A -85,B 0,C 180,E1 4850.496,E2 4850.496} C_VEL
LIN {X 0,Y 166.457,Z 946.833,A -85,B 0,C 180,E1 4848.215,E2 4848.215} C_VEL
LIN {X 0,Y 155.977,Z 957.308,A -85,B 0,C 180,E1 4845.454,E2 4845.454} C_VEL
LIN {X 0,Y 144.239,Z 967.082,A -85,B 0,C 180,E1 4841.745,E2 4841.745} C_VEL
LIN {X 0,Y 133.171,Z 974.657,A -85,B 0,C 180,E1 4837.442,E2 4837.442} C_VEL
LIN {X 0,Y 122.251,Z 980.683,A -85,B 0,C 180,E1 4832.042,E2 4832.042} C_VEL
LIN {X 0,Y 111.984,Z 985.118,A -85,B 0,C 180,E1 4825.227,E2 4825.227} C_VEL
LIN {X 0,Y 103.512,Z 987.567,A -85,B 0,C 180,E1 4817.231,E2 4817.231} C_VEL
LIN {X 0,Y 96.864,Z 988.185,A -85,B 0,C 180,E1 4807.36,E2 4807.36} C_VEL
LIN {X 0,Y 93.255,Z 986.9,A -85,B 0,C 180,E1 4797.136,E2 4797.136} C_VEL
LIN {X 0,Y 92.304,Z 983.73,A -85,B 0,C 180,E1 4786.357,E2 4786.357} C_VEL
LIN {X 0,Y 93.9,Z 978.887,A -85,B 0,C 180,E1 4776.111,E2 4776.111} C_VEL
LIN {X 0,Y 97.548,Z 972.517,A -85,B 0,C 180,E1 4767.061,E2 4767.061} C_VEL
LIN {X 0,Y 103.116,Z 964.229,A -85,B 0,C 180,E1 4758.817,E2 4758.817} C_VEL
LIN {X 0,Y 109.304,Z 955.184,A -85,B 0,C 180,E1 4752.429,E2 4752.429} C_VEL
LIN {X 0,Y 116.533,Z 943.926,A -85,B 0,C 180,E1 4746.753,E2 4746.753} C_VEL
LIN {X 0,Y 123.949,Z 931.135,A -85,B 0,C 180,E1 4742.103,E2 4742.103} C_VEL
LIN {X 0,Y 130.582,Z 917.888,A -85,B 0,C 180,E1 4738.621,E2 4738.621} C_VEL
LIN {X 0,Y 136.865,Z 902.984,A -85,B 0,C 180,E1 4735.769,E2 4735.769} C_VEL
LIN {X 0,Y 141.876,Z 888.271,A -85,B 0,C 180,E1 4733.701,E2 4733.701} C_VEL
LIN {X 0,Y 146.111,Z 871.626,A -85,B 0,C 180,E1 4732.045,E2 4732.045} C_VEL
LIN {X 0,Y 149.109,Z 854.074,A -85,B 0,C 180,E1 4730.878,E2 4730.878} C_VEL
LIN {X 0,Y 155.589,Z 787.857,A -85,B 0,C 180,E1 4728.603,E2 4728.603} C_VEL
LIN {X 0,Y 156.954,Z 772.709,A -85,B 0,C 180,E1 4728.066,E2 4728.066} C_VEL
LIN {X 0,Y 156.62,Z 757.076,A -85,B 0,C 180,E1 4726.435,E2 4726.435} C_VEL
LIN {X 0,Y 152.263,Z 745.635,A -85,B 0,C 180,E1 4722.18,E2 4722.18} C_VEL
LIN {X 0,Y 148.731,Z 737.702,A -85,B 0,C 180,E1 4718.135,E2 4718.135} C_VEL
LIN {X 0,Y 145.226,Z 730.355,A -85,B 0,C 180,E1 4713.186,E2 4713.186} C_VEL
LIN {X 0,Y 142.059,Z 724.251,A -85,B 0,C 180,E1 4706.774,E2 4706.774} C_VEL
LIN {X 0,Y 140.917,Z 722.384,A -85,B 0,C 180,E1 4703.413,E2 4703.413} C_VEL
LIN {X 0,Y 139.976,Z 720.126,A -85,B 0,C 180,E1 4697.459,E2 4697.459} C_VEL
LIN {X 0,Y 140.391,Z 720.351,A -85,B 0,C 180,E1 4690.257,E2 4690.257} C_VEL
LIN {X 0,Y 141.256,Z 721.507,A -85,B 0,C 180,E1 4686.708,E2 4686.708} C_VEL
LIN {X 0,Y 143.409,Z 724.566,A -85,B 0,C 180,E1 4681.399,E2 4681.399} C_VEL
LIN {X 0,Y 146.474,Z 729.595,A -85,B 0,C 180,E1 4676.185,E2 4676.185} C_VEL
LIN {X 0,Y 149.952,Z 735.685,A -85,B 0,C 180,E1 4671.759,E2 4671.759} C_VEL
LIN {X 0,Y 153.927,Z 743.408,A -85,B 0,C 180,E1 4667.575,E2 4667.575} C_VEL
LIN {X 0,Y 158.137,Z 752.717,A -85,B 0,C 180,E1 4663.801,E2 4663.801} C_VEL
LIN {X 0,Y 161.183,Z 760.347,A -85,B 0,C 180,E1 4661.352,E2 4661.352} C_VEL
LIN {X 0,Y 150.963,Z 868.522,A -85,B 0,C 180,E1 4657.95,E2 4657.95} C_VEL
LIN {X 0,Y 147.699,Z 886.639,A -85,B 0,C 180,E1 4656.914,E2 4656.914} C_VEL
LIN {X 0,Y 143.149,Z 903.455,A -85,B 0,C 180,E1 4655.519,E2 4655.519} C_VEL
LIN {X 0,Y 137.311,Z 919.744,A -85,B 0,C 180,E1 4653.594,E2 4653.594} C_VEL
LIN {X 0,Y 130.383,Z 935.402,A -85,B 0,C 180,E1 4650.956,E2 4650.956} C_VEL
LIN {X 0,Y 122.831,Z 949.983,A -85,B 0,C 180,E1 4647.505,E2 4647.505} C_VEL
LIN {X 0,Y 115.02,Z 963.307,A -85,B 0,C 180,E1 4643.108,E2 4643.108} C_VEL
LIN {X 0,Y 107.223,Z 975.45,A -85,B 0,C 180,E1 4637.451,E2 4637.451} C_VEL
LIN {X 0,Y 100.233,Z 986.127,A -85,B 0,C 180,E1 4630.422,E2 4630.422} C_VEL
LIN {X 0,Y 94.629,Z 995.34,A -85,B 0,C 180,E1 4621.893,E2 4621.893} C_VEL
LIN {X 0,Y 91.126,Z 1003.013,A -85,B 0,C 180,E1 4611.906,E2 4611.906} C_VEL
LIN {X 0,Y 90.358,Z 1008.676,A -85,B 0,C 180,E1 4601.49,E2 4601.49} C_VEL
LIN {X 0,Y 92.005,Z 1012.533,A -85,B 0,C 180,E1 4591.189,E2 4591.189} C_VEL
LIN {X 0,Y 92.218,Z 1012.994,A -85,B 0,C 180,E1 4589.38,E2 4589.38} C_VEL
LIN {X 0,Y 90.093,Z 1013.808,A -85,B 0,C 180,E1 4578.478,E2 4578.478} C_VEL
LIN {X 0,Y 90.608,Z 1013.204,A -85,B 0,C 180,E1 4568.934,E2 4568.934} C_VEL
LIN {X 0,Y 90.833,Z 1012.417,A -85,B 0,C 180,E1 4564.053,E2 4564.053} C_VEL
LIN {X 0,Y 90.945,Z 1008.926,A -85,B 0,C 180,E1 4551.519,E2 4551.519} C_VEL
LIN {X 0,Y 93.423,Z 1007.147,A -85,B 0,C 180,E1 4547.074,E2 4547.074} C_VEL
LIN {X 0,Y 103.986,Z 1001.76,A -85,B 0,C 180,E1 4537.96,E2 4537.96} C_VEL
LIN {X 0,Y 116.054,Z 994.799,A -85,B 0,C 180,E1 4531.125,E2 4531.125} C_VEL
LIN {X 0,Y 128.19,Z 986.748,A -85,B 0,C 180,E1 4526.238,E2 4526.238} C_VEL
LIN {X 0,Y 140.644,Z 977.149,A -85,B 0,C 180,E1 4522.455,E2 4522.455} C_VEL
LIN {X 0,Y 153.588,Z 965.435,A -85,B 0,C 180,E1 4519.39,E2 4519.39} C_VEL
LIN {X 0,Y 165.345,Z 952.859,A -85,B 0,C 180,E1 4517.169,E2 4517.169} C_VEL
LIN {X 0,Y 175.896,Z 939.393,A -85,B 0,C 180,E1 4515.528,E2 4515.528} C_VEL
LIN {X 0,Y 185.217,Z 924.992,A -85,B 0,C 180,E1 4514.305,E2 4514.305} C_VEL
LIN {X 0,Y 193.703,Z 908.767,A -85,B 0,C 180,E1 4513.345,E2 4513.345} C_VEL
LIN {X 0,Y 200.34,Z 892.423,A -85,B 0,C 180,E1 4512.657,E2 4512.657} C_VEL
LIN {X 0,Y 205.399,Z 875.013,A -85,B 0,C 180,E1 4512.127,E2 4512.127} C_VEL
LIN {X 0,Y 208.754,Z 856.728,A -85,B 0,C 180,E1 4511.711,E2 4511.711} C_VEL
LIN {X 0,Y 214.482,Z 809.245,A -85,B 0,C 180,E1 4510.746,E2 4510.746} C_VEL
LIN {X 0,Y 213.873,Z 807.872,A -85,B 0,C 180,E1 4508.332,E2 4508.332} C_VEL
LIN {X 0,Y 213.443,Z 807.645,A -85,B 0,C 180,E1 4504.567,E2 4504.567} C_VEL
LIN {X 0,Y 213.77,Z 810.07,A -85,B 0,C 180,E1 4500.669,E2 4500.669} C_VEL
LIN {X 0,Y 213.876,Z 811.262,A -85,B 0,C 180,E1 4499.845,E2 4499.845} C_VEL
LIN {X 0,Y 207.797,Z 859.24,A -85,B 0,C 180,E1 4498.799,E2 4498.799} C_VEL
LIN {X 0,Y 204.008,Z 876.269,A -85,B 0,C 180,E1 4498.152,E2 4498.152} C_VEL
LIN {X 0,Y 198.694,Z 892.468,A -85,B 0,C 180,E1 4497.288,E2 4497.288} C_VEL
LIN {X 0,Y 191.875,Z 907.906,A -85,B 0,C 180,E1 4496.174,E2 4496.174} C_VEL
LIN {X 0,Y 183.736,Z 922.266,A -85,B 0,C 180,E1 4494.779,E2 4494.779} C_VEL
LIN {X 0,Y 174.27,Z 935.809,A -85,B 0,C 180,E1 4493.009,E2 4493.009} C_VEL
LIN {X 0,Y 164.057,Z 947.801,A -85,B 0,C 180,E1 4490.865,E2 4490.865} C_VEL
LIN {X 0,Y 153.191,Z 958.316,A -85,B 0,C 180,E1 4488.245,E2 4488.245} C_VEL
LIN {X 0,Y 140.973,Z 968.105,A -85,B 0,C 180,E1 4484.706,E2 4484.706} C_VEL
LIN {X 0,Y 129.362,Z 975.719,A -85,B 0,C 180,E1 4480.553,E2 4480.553} C_VEL
LIN {X 0,Y 117.783,Z 981.776,A -85,B 0,C 180,E1 4475.273,E2 4475.273} C_VEL
LIN {X 0,Y 106.731,Z 986.236,A -85,B 0,C 180,E1 4468.482,E2 4468.482} C_VEL
LIN {X 0,Y 97.43,Z 988.747,A -85,B 0,C 180,E1 4460.323,E2 4460.323} C_VEL
LIN {X 0,Y 89.999,Z 989.42,A -85,B 0,C 180,E1 4450.116,E2 4450.116} C_VEL
LIN {X 0,Y 85.755,Z 988.28,A -85,B 0,C 180,E1 4439.32,E2 4439.32} C_VEL
LIN {X 0,Y 84.34,Z 985.35,A -85,B 0,C 180,E1 4427.952,E2 4427.952} C_VEL
LIN {X 0,Y 85.693,Z 980.675,A -85,B 0,C 180,E1 4416.699,E2 4416.699} C_VEL
LIN {X 0,Y 89.358,Z 974.575,A -85,B 0,C 180,E1 4406.792,E2 4406.792} C_VEL
LIN {X 0,Y 95.116,Z 966.504,A -85,B 0,C 180,E1 4397.86,E2 4397.86} C_VEL
LIN {X 0,Y 102.113,Z 956.984,A -85,B 0,C 180,E1 4390.553,E2 4390.553} C_VEL
LIN {X 0,Y 109.741,Z 945.941,A -85,B 0,C 180,E1 4384.644,E2 4384.644} C_VEL
LIN {X 0,Y 117.872,Z 932.77,A -85,B 0,C 180,E1 4379.686,E2 4379.686} C_VEL
LIN {X 0,Y 124.83,Z 919.745,A -85,B 0,C 180,E1 4376.172,E2 4376.172} C_VEL
LIN {X 0,Y 131.396,Z 905.058,A -85,B 0,C 180,E1 4373.318,E2 4373.318} C_VEL
LIN {X 0,Y 136.998,Z 889.509,A -85,B 0,C 180,E1 4371.121,E2 4371.121} C_VEL
LIN {X 0,Y 141.42,Z 873.109,A -85,B 0,C 180,E1 4369.49,E2 4369.49} C_VEL
LIN {X 0,Y 144.643,Z 855.291,A -85,B 0,C 180,E1 4368.307,E2 4368.307} C_VEL
LIN {X 0,Y 150.308,Z 799.811,A -85,B 0,C 180,E1 4366.389,E2 4366.389} C_VEL
LIN {X 0,Y 152.848,Z 773.707,A -85,B 0,C 180,E1 4365.533,E2 4365.533} C_VEL
LIN {X 0,Y 152.7,Z 761.021,A -85,B 0,C 180,E1 4364.15,E2 4364.15} C_VEL
LIN {X 0,Y 149.26,Z 751.348,A -85,B 0,C 180,E1 4360.337,E2 4360.337} C_VEL
LIN {X 0,Y 145.902,Z 743.181,A -85,B 0,C 180,E1 4356.003,E2 4356.003} C_VEL
LIN {X 0,Y 142.892,Z 736.568,A -85,B 0,C 180,E1 4351.069,E2 4351.069} C_VEL
LIN {X 0,Y 140.472,Z 731.387,A -85,B 0,C 180,E1 4345.283,E2 4345.283} C_VEL
LIN {X 0,Y 138.96,Z 728.04,A -85,B 0,C 180,E1 4337.159,E2 4337.159} C_VEL
LIN {X 0,Y 139.453,Z 728.365,A -85,B 0,C 180,E1 4329.909,E2 4329.909} C_VEL
LIN {X 0,Y 140.692,Z 730.277,A -85,B 0,C 180,E1 4325.302,E2 4325.302} C_VEL
LIN {X 0,Y 142.14,Z 732.567,A -85,B 0,C 180,E1 4321.815,E2 4321.815} C_VEL
LIN {X 0,Y 144.714,Z 737.045,A -85,B 0,C 180,E1 4317.13,E2 4317.13} C_VEL
LIN {X 0,Y 147.847,Z 742.946,A -85,B 0,C 180,E1 4312.814,E2 4312.814} C_VEL
LIN {X 0,Y 151.494,Z 750.66,A -85,B 0,C 180,E1 4308.677,E2 4308.677} C_VEL
LIN {X 0,Y 155.204,Z 759.462,A -85,B 0,C 180,E1 4305.068,E2 4305.068} C_VEL
LIN {X 0,Y 156.682,Z 763.719,A -85,B 0,C 180,E1 4303.715,E2 4303.715} C_VEL
LIN {X 0,Y 146.446,Z 867.882,A -85,B 0,C 180,E1 4300.5,E2 4300.5} C_VEL
LIN {X 0,Y 143.057,Z 886.056,A -85,B 0,C 180,E1 4299.484,E2 4299.484} C_VEL
LIN {X 0,Y 138.222,Z 903.276,A -85,B 0,C 180,E1 4298.085,E2 4298.085} C_VEL
LIN {X 0,Y 132.216,Z 919.313,A -85,B 0,C 180,E1 4296.214,E2 4296.214} C_VEL
LIN {X 0,Y 125.012,Z 934.908,A -85,B 0,C 180,E1 4293.613,E2 4293.613} C_VEL
LIN {X 0,Y 117.097,Z 949.463,A -85,B 0,C 180,E1 4290.166,E2 4290.166} C_VEL
LIN {X 0,Y 108.892,Z 962.698,A -85,B 0,C 180,E1 4285.732,E2 4285.732} C_VEL
LIN {X 0,Y 100.616,Z 974.754,A -85,B 0,C 180,E1 4279.925,E2 4279.925} C_VEL
LIN {X 0,Y 92.649,Z 986.05,A -85,B 0,C 180,E1 4272,E2 4272} C_VEL
LIN {X 0,Y 86.622,Z 995.253,A -85,B 0,C 180,E1 4262.584,E2 4262.584} C_VEL
LIN {X 0,Y 83.106,Z 1002.485,A -85,B 0,C 180,E1 4251.9,E2 4251.9} C_VEL
LIN {X 0,Y 82.531,Z 1008.255,A -85,B 0,C 180,E1 4239.766,E2 4239.766} C_VEL
LIN {X 0,Y 84.312,Z 1011.531,A -85,B 0,C 180,E1 4229.662,E2 4229.662} C_VEL
LIN {X 0,Y 82.138,Z 1012.488,A -85,B 0,C 180,E1 4217.344,E2 4217.344} C_VEL
LIN {X 0,Y 83.608,Z 1011.716,A -85,B 0,C 180,E1 4204.501,E2 4204.501} C_VEL
LIN {X 0,Y 89.062,Z 1009.228,A -85,B 0,C 180,E1 4192.683,E2 4192.683} C_VEL
LIN {X 0,Y 93.423,Z 1007.147,A -85,B 0,C 180,E1 4187.074,E2 4187.074} C_VEL
LIN {X 0,Y 96.427,Z 1005.226,A -85,B 0,C 180,E1 4182.916,E2 4182.916} C_VEL
LIN {X 0,Y 103.233,Z 999.215,A -85,B 0,C 180,E1 4172.588,E2 4172.588} C_VEL
LIN {X 0,Y 107.734,Z 996.441,A -85,B 0,C 180,E1 4169.489,E2 4169.489} C_VEL
LIN {X 0,Y 120.623,Z 988.829,A -85,B 0,C 180,E1 4164.246,E2 4164.246} C_VEL
LIN {X 0,Y 134.238,Z 979.349,A -85,B 0,C 180,E1 4160.2,E2 4160.2} C_VEL
LIN {X 0,Y 147.56,Z 968.361,A -85,B 0,C 180,E1 4157.176,E2 4157.176} C_VEL
LIN {X 0,Y 159.998,Z 956.147,A -85,B 0,C 180,E1 4154.953,E2 4154.953} C_VEL
LIN {X 0,Y 171.562,Z 942.463,A -85,B 0,C 180,E1 4153.278,E2 4153.278} C_VEL
LIN {X 0,Y 181.973,Z 927.542,A -85,B 0,C 180,E1 4152.035,E2 4152.035} C_VEL
LIN {X 0,Y 190.579,Z 912.321,A -85,B 0,C 180,E1 4151.164,E2 4151.164} C_VEL
LIN {X 0,Y 197.786,Z 895.968,A -85,B 0,C 180,E1 4150.504,E2 4150.504} C_VEL
LIN {X 0,Y 203.494,Z 878.488,A -85,B 0,C 180,E1 4149.99,E2 4149.99} C_VEL
LIN {X 0,Y 207.259,Z 861.016,A -85,B 0,C 180,E1 4149.602,E2 4149.602} C_VEL
LIN {X 0,Y 212.949,Z 815.935,A -85,B 0,C 180,E1 4148.777,E2 4148.777} C_VEL
LIN {X 0,Y 212.43,Z 815.518,A -85,B 0,C 180,E1 4144.859,E2 4144.859} C_VEL
LIN {X 0,Y 212.525,Z 817.334,A -85,B 0,C 180,E1 4141.881,E2 4141.881} C_VEL
LIN {X 0,Y 206.916,Z 860.343,A -85,B 0,C 180,E1 4140.977,E2 4140.977} C_VEL
LIN {X 0,Y 203.006,Z 877.385,A -85,B 0,C 180,E1 4140.365,E2 4140.365} C_VEL
LIN {X 0,Y 197.478,Z 893.763,A -85,B 0,C 180,E1 4139.545,E2 4139.545} C_VEL
LIN {X 0,Y 190.401,Z 909.275,A -85,B 0,C 180,E1 4138.495,E2 4138.495} C_VEL
LIN {X 0,Y 181.854,Z 923.891,A -85,B 0,C 180,E1 4137.163,E2 4137.163} C_VEL
LIN {X 0,Y 172.008,Z 937.477,A -85,B 0,C 180,E1 4135.488,E2 4135.488} C_VEL
LIN {X 0,Y 161.519,Z 949.285,A -85,B 0,C 180,E1 4133.486,E2 4133.486} C_VEL
LIN {X 0,Y 149.859,Z 960.095,A -85,B 0,C 180,E1 4130.912,E2 4130.912} C_VEL
LIN {X 0,Y 138.1,Z 969.128,A -85,B 0,C 180,E1 4127.797,E2 4127.797} C_VEL
LIN {X 0,Y 125.957,Z 976.778,A -85,B 0,C 180,E1 4123.843,E2 4123.843} C_VEL
LIN {X 0,Y 113.72,Z 982.87,A -85,B 0,C 180,E1 4118.744,E2 4118.744} C_VEL
LIN {X 0,Y 101.86,Z 987.363,A -85,B 0,C 180,E1 4112.058,E2 4112.058} C_VEL
LIN {X 0,Y 91.672,Z 989.938,A -85,B 0,C 180,E1 4103.813,E2 4103.813} C_VEL
LIN {X 0,Y 83.702,Z 990.665,A -85,B 0,C 180,E1 4093.853,E2 4093.853} C_VEL
LIN {X 0,Y 78.293,Z 989.572,A -85,B 0,C 180,E1 4081.573,E2 4081.573} C_VEL
LIN {X 0,Y 76.419,Z 986.727,A -85,B 0,C 180,E1 4069.091,E2 4069.091} C_VEL
LIN {X 0,Y 77.655,Z 982.118,A -85,B 0,C 180,E1 4056.653,E2 4056.653} C_VEL
LIN {X 0,Y 81.491,Z 976.112,A -85,B 0,C 180,E1 4045.777,E2 4045.777} C_VEL
LIN {X 0,Y 87.614,Z 968.174,A -85,B 0,C 180,E1 4036.133,E2 4036.133} C_VEL
LIN {X 0,Y 95.049,Z 958.771,A -85,B 0,C 180,E1 4028.395,E2 4028.395} C_VEL
LIN {X 0,Y 103.118,Z 947.954,A -85,B 0,C 180,E1 4022.261,E2 4022.261} C_VEL
LIN {X 0,Y 111.318,Z 935.555,A -85,B 0,C 180,E1 4017.388,E2 4017.388} C_VEL
LIN {X 0,Y 119.329,Z 921.556,A -85,B 0,C 180,E1 4013.492,E2 4013.492} C_VEL
LIN {X 0,Y 126.186,Z 907.132,A -85,B 0,C 180,E1 4010.661,E2 4010.661} C_VEL
LIN {X 0,Y 132.419,Z 890.745,A -85,B 0,C 180,E1 4008.358,E2 4008.358} C_VEL
LIN {X 0,Y 137.078,Z 874.377,A -85,B 0,C 180,E1 4006.748,E2 4006.748} C_VEL
LIN {X 0,Y 140.512,Z 856.349,A -85,B 0,C 180,E1 4005.57,E2 4005.57} C_VEL
LIN {X 0,Y 145.717,Z 807.468,A -85,B 0,C 180,E1 4003.891,E2 4003.891} C_VEL
LIN {X 0,Y 149.057,Z 774.716,A -85,B 0,C 180,E1 4002.867,E2 4002.867} C_VEL
LIN {X 0,Y 149.058,Z 765.013,A -85,B 0,C 180,E1 4001.774,E2 4001.774} C_VEL
LIN {X 0,Y 146.015,Z 756.066,A -85,B 0,C 180,E1 3997.922,E2 3997.922} C_VEL
LIN {X 0,Y 143.15,Z 748.601,A -85,B 0,C 180,E1 3993.611,E2 3993.611} C_VEL
LIN {X 0,Y 141.127,Z 743.698,A -85,B 0,C 180,E1 3989.733,E2 3989.733} C_VEL
LIN {X 0,Y 139.156,Z 738.982,A -85,B 0,C 180,E1 3984.404,E2 3984.404} C_VEL
LIN {X 0,Y 137.946,Z 735.955,A -85,B 0,C 180,E1 3976.855,E2 3976.855} C_VEL
LIN {X 0,Y 138.52,Z 736.387,A -85,B 0,C 180,E1 3969.557,E2 3969.557} C_VEL
LIN {X 0,Y 140.451,Z 739.607,A -85,B 0,C 180,E1 3963.266,E2 3963.266} C_VEL
LIN {X 0,Y 142.941,Z 744.377,A -85,B 0,C 180,E1 3958.197,E2 3958.197} C_VEL
LIN {X 0,Y 145.734,Z 750.104,A -85,B 0,C 180,E1 3953.975,E2 3953.975} C_VEL
LIN {X 0,Y 149.324,Z 758.367,A -85,B 0,C 180,E1 3949.585,E2 3949.585} C_VEL
LIN {X 0,Y 152.494,Z 766.729,A -85,B 0,C 180,E1 3946.223,E2 3946.223} C_VEL
LIN {X 0,Y 142.235,Z 867.243,A -85,B 0,C 180,E1 3943.204,E2 3943.204} C_VEL
LIN {X 0,Y 138.729,Z 885.402,A -85,B 0,C 180,E1 3942.223,E2 3942.223} C_VEL
LIN {X 0,Y 133.849,Z 902.255,A -85,B 0,C 180,E1 3940.906,E2 3940.906} C_VEL
LIN {X 0,Y 127.842,Z 917.885,A -85,B 0,C 180,E1 3939.169,E2 3939.169} C_VEL
LIN {X 0,Y 120.342,Z 933.581,A -85,B 0,C 180,E1 3936.651,E2 3936.651} C_VEL
LIN {X 0,Y 111.977,Z 948.318,A -85,B 0,C 180,E1 3933.244,E2 3933.244} C_VEL
LIN {X 0,Y 103.379,Z 961.492,A -85,B 0,C 180,E1 3928.867,E2 3928.867} C_VEL
LIN {X 0,Y 94.858,Z 973.183,A -85,B 0,C 180,E1 3923.236,E2 3923.236} C_VEL
LIN {X 0,Y 86.684,Z 983.893,A -85,B 0,C 180,E1 3915.657,E2 3915.657} C_VEL
LIN {X 0,Y 79.924,Z 993.122,A -85,B 0,C 180,E1 3906.015,E2 3906.015} C_VEL
LIN {X 0,Y 75.542,Z 1000.781,A -85,B 0,C 180,E1 3894.226,E2 3894.226} C_VEL
LIN {X 0,Y 74.473,Z 1006.471,A -85,B 0,C 180,E1 3881.463,E2 3881.463} C_VEL
LIN {X 0,Y 76.297,Z 1010.121,A -85,B 0,C 180,E1 3869.626,E2 3869.626} C_VEL
LIN {X 0,Y 74.214,Z 1011.167,A -85,B 0,C 180,E1 3855.931,E2 3855.931} C_VEL
LIN {X 0,Y 76.546,Z 1010.414,A -85,B 0,C 180,E1 3841.062,E2 3841.062} C_VEL
LIN {X 0,Y 83.137,Z 1007.954,A -85,B 0,C 180,E1 3828.59,E2 3828.59} C_VEL
LIN {X 0,Y 93.158,Z 1003.683,A -85,B 0,C 180,E1 3818.419,E2 3818.419} C_VEL
LIN {X 0,Y 105.633,Z 997.537,A -85,B 0,C 180,E1 3810.532,E2 3810.532} C_VEL
LIN {X 0,Y 107.734,Z 996.441,A -85,B 0,C 180,E1 3809.489,E2 3809.489} C_VEL
LIN {X 0,Y 112.502,Z 993.51,A -85,B 0,C 180,E1 3806.684,E2 3806.684} C_VEL
LIN {X 0,Y 123.178,Z 984.921,A -85,B 0,C 180,E1 3799.514,E2 3799.514} C_VEL
LIN {X 0,Y 128.476,Z 981.064,A -85,B 0,C 180,E1 3797.622,E2 3797.622} C_VEL
LIN {X 0,Y 141.678,Z 971.11,A -85,B 0,C 180,E1 3794.797,E2 3794.797} C_VEL
LIN {X 0,Y 154.713,Z 959.311,A -85,B 0,C 180,E1 3792.616,E2 3792.616} C_VEL
LIN {X 0,Y 167.03,Z 945.963,A -85,B 0,C 180,E1 3790.974,E2 3790.974} C_VEL
LIN {X 0,Y 177.581,Z 932.161,A -85,B 0,C 180,E1 3789.829,E2 3789.829} C_VEL
LIN {X 0,Y 186.768,Z 917.368,A -85,B 0,C 180,E1 3788.992,E2 3788.992} C_VEL
LIN {X 0,Y 194.482,Z 901.774,A -85,B 0,C 180,E1 3788.375,E2 3788.375} C_VEL
LIN {X 0,Y 200.872,Z 884.86,A -85,B 0,C 180,E1 3787.888,E2 3787.888} C_VEL
LIN {X 0,Y 205.421,Z 867.582,A -85,B 0,C 180,E1 3787.512,E2 3787.512} C_VEL
LIN {X 0,Y 208.678,Z 846.3,A -85,B 0,C 180,E1 3787.136,E2 3787.136} C_VEL
LIN {X 0,Y 211.555,Z 823.473,A -85,B 0,C 180,E1 3786.724,E2 3786.724} C_VEL
LIN {X 0,Y 211.379,Z 823.659,A -85,B 0,C 180,E1 3784.612,E2 3784.612} C_VEL
LIN {X 0,Y 211.341,Z 824.219,A -85,B 0,C 180,E1 3783.926,E2 3783.926} C_VEL
LIN {X 0,Y 206.346,Z 861.4,A -85,B 0,C 180,E1 3783.172,E2 3783.172} C_VEL
LIN {X 0,Y 202.303,Z 878.521,A -85,B 0,C 180,E1 3782.596,E2 3782.596} C_VEL
LIN {X 0,Y 196.571,Z 895.058,A -85,B 0,C 180,E1 3781.826,E2 3781.826} C_VEL
LIN {X 0,Y 189.495,Z 910.184,A -85,B 0,C 180,E1 3780.882,E2 3780.882} C_VEL
LIN {X 0,Y 180.912,Z 924.589,A -85,B 0,C 180,E1 3779.683,E2 3779.683} C_VEL
LIN {X 0,Y 171.061,Z 937.943,A -85,B 0,C 180,E1 3778.187,E2 3778.187} C_VEL
LIN {X 0,Y 160.301,Z 949.886,A -85,B 0,C 180,E1 3776.355,E2 3776.355} C_VEL
LIN {X 0,Y 148.767,Z 960.38,A -85,B 0,C 180,E1 3774.098,E2 3774.098} C_VEL
LIN {X 0,Y 135.648,Z 970.173,A -85,B 0,C 180,E1 3771.007,E2 3771.007} C_VEL
LIN {X 0,Y 122.99,Z 977.832,A -85,B 0,C 180,E1 3767.301,E2 3767.301} C_VEL
LIN {X 0,Y 110.105,Z 983.961,A -85,B 0,C 180,E1 3762.457,E2 3762.457} C_VEL
LIN {X 0,Y 97.426,Z 988.49,A -85,B 0,C 180,E1 3755.976,E2 3755.976} C_VEL
LIN {X 0,Y 86.3,Z 991.126,A -85,B 0,C 180,E1 3747.753,E2 3747.753} C_VEL
LIN {X 0,Y 77.335,Z 991.901,A -85,B 0,C 180,E1 3737.47,E2 3737.47} C_VEL
LIN {X 0,Y 70.977,Z 990.854,A -85,B 0,C 180,E1 3724.295,E2 3724.295} C_VEL
LIN {X 0,Y 68.529,Z 988.093,A -85,B 0,C 180,E1 3710.496,E2 3710.496} C_VEL
LIN {X 0,Y 69.613,Z 983.55,A -85,B 0,C 180,E1 3696.597,E2 3696.597} C_VEL
LIN {X 0,Y 74.018,Z 977.183,A -85,B 0,C 180,E1 3683.795,E2 3683.795} C_VEL
LIN {X 0,Y 80.721,Z 969.226,A -85,B 0,C 180,E1 3673.446,E2 3673.446} C_VEL
LIN {X 0,Y 88.762,Z 959.819,A -85,B 0,C 180,E1 3665.367,E2 3665.367} C_VEL
LIN {X 0,Y 97.392,Z 949.004,A -85,B 0,C 180,E1 3659.113,E2 3659.113} C_VEL
LIN {X 0,Y 106.078,Z 936.615,A -85,B 0,C 180,E1 3654.239,E2 3654.239} C_VEL
LIN {X 0,Y 114.503,Z 922.641,A -85,B 0,C 180,E1 3650.397,E2 3650.397} C_VEL
LIN {X 0,Y 121.674,Z 908.286,A -85,B 0,C 180,E1 3647.635,E2 3647.635} C_VEL
LIN {X 0,Y 128.17,Z 891.982,A -85,B 0,C 180,E1 3645.403,E2 3645.403} C_VEL
LIN {X 0,Y 133.097,Z 875.536,A -85,B 0,C 180,E1 3643.827,E2 3643.827} C_VEL
LIN {X 0,Y 136.647,Z 857.876,A -85,B 0,C 180,E1 3642.699,E2 3642.699} C_VEL
LIN {X 0,Y 140.368,Z 824.761,A -85,B 0,C 180,E1 3641.51,E2 3641.51} C_VEL
LIN {X 0,Y 145.603,Z 775.804,A -85,B 0,C 180,E1 3640.076,E2 3640.076} C_VEL
LIN {X 0,Y 145.659,Z 769.188,A -85,B 0,C 180,E1 3639.291,E2 3639.291} C_VEL
LIN {X 0,Y 143.279,Z 761.564,A -85,B 0,C 180,E1 3635.826,E2 3635.826} C_VEL
LIN {X 0,Y 140.971,Z 754.942,A -85,B 0,C 180,E1 3631.779,E2 3631.779} C_VEL
LIN {X 0,Y 139.484,Z 750.926,A -85,B 0,C 180,E1 3628.47,E2 3628.47} C_VEL
LIN {X 0,Y 137.819,Z 746.435,A -85,B 0,C 180,E1 3623.291,E2 3623.291} C_VEL
LIN {X 0,Y 136.935,Z 743.871,A -85,B 0,C 180,E1 3616.546,E2 3616.546} C_VEL
LIN {X 0,Y 137.501,Z 744.332,A -85,B 0,C 180,E1 3609.629,E2 3609.629} C_VEL
LIN {X 0,Y 139.054,Z 747.221,A -85,B 0,C 180,E1 3604.124,E2 3604.124} C_VEL
LIN {X 0,Y 141.217,Z 751.709,A -85,B 0,C 180,E1 3599.291,E2 3599.291} C_VEL
LIN {X 0,Y 143.654,Z 757.212,A -85,B 0,C 180,E1 3595.21,E2 3595.21} C_VEL
LIN {X 0,Y 146.799,Z 765.072,A -85,B 0,C 180,E1 3590.988,E2 3590.988} C_VEL
LIN {X 0,Y 148.549,Z 770.368,A -85,B 0,C 180,E1 3588.85,E2 3588.85} C_VEL
LIN {X 0,Y 138.341,Z 866.71,A -85,B 0,C 180,E1 3586.064,E2 3586.064} C_VEL
LIN {X 0,Y 134.689,Z 884.939,A -85,B 0,C 180,E1 3585.119,E2 3585.119} C_VEL
LIN {X 0,Y 129.786,Z 901.341,A -85,B 0,C 180,E1 3583.899,E2 3583.899} C_VEL
LIN {X 0,Y 123.393,Z 917.401,A -85,B 0,C 180,E1 3582.199,E2 3582.199} C_VEL
LIN {X 0,Y 115.493,Z 933.242,A -85,B 0,C 180,E1 3579.74,E2 3579.74} C_VEL
LIN {X 0,Y 106.878,Z 947.699,A -85,B 0,C 180,E1 3576.467,E2 3576.467} C_VEL
LIN {X 0,Y 97.829,Z 960.804,A -85,B 0,C 180,E1 3572.14,E2 3572.14} C_VEL
LIN {X 0,Y 88.771,Z 972.427,A -85,B 0,C 180,E1 3566.461,E2 3566.461} C_VEL
LIN {X 0,Y 79.703,Z 983.397,A -85,B 0,C 180,E1 3558.329,E2 3558.329} C_VEL
LIN {X 0,Y 72.487,Z 992.368,A -85,B 0,C 180,E1 3548.167,E2 3548.167} C_VEL
LIN {X 0,Y 67.716,Z 999.834,A -85,B 0,C 180,E1 3535.355,E2 3535.355} C_VEL
LIN {X 0,Y 66.539,Z 1005.411,A -85,B 0,C 180,E1 3521.267,E2 3521.267} C_VEL
LIN {X 0,Y 68.262,Z 1008.702,A -85,B 0,C 180,E1 3509.582,E2 3509.582} C_VEL
LIN {X 0,Y 66.339,Z 1009.841,A -85,B 0,C 180,E1 3494.26,E2 3494.26} C_VEL
LIN {X 0,Y 69.469,Z 1009.196,A -85,B 0,C 180,E1 3477.825,E2 3477.825} C_VEL
LIN {X 0,Y 77.704,Z 1006.678,A -85,B 0,C 180,E1 3463.899,E2 3463.899} C_VEL
LIN {X 0,Y 88.981,Z 1002.431,A -85,B 0,C 180,E1 3453.747,E2 3453.747} C_VEL
LIN {X 0,Y 102.507,Z 996.321,A -85,B 0,C 180,E1 3446.187,E2 3446.187} C_VEL
LIN {X 0,Y 116.643,Z 988.669,A -85,B 0,C 180,E1 3440.88,E2 3440.88} C_VEL
LIN {X 0,Y 128.476,Z 981.064,A -85,B 0,C 180,E1 3437.622,E2 3437.622} C_VEL
LIN {X 0,Y 133.845,Z 977.034,A -85,B 0,C 180,E1 3435.912,E2 3435.912} C_VEL
LIN {X 0,Y 145.802,Z 965.959,A -85,B 0,C 180,E1 3431.083,E2 3431.083} C_VEL
LIN {X 0,Y 151.046,Z 961.066,A -85,B 0,C 180,E1 3429.94,E2 3429.94} C_VEL
LIN {X 0,Y 163.269,Z 948.716,A -85,B 0,C 180,E1 3428.498,E2 3428.498} C_VEL
LIN {X 0,Y 174.439,Z 934.988,A -85,B 0,C 180,E1 3427.43,E2 3427.43} C_VEL
LIN {X 0,Y 184.217,Z 920.299,A -85,B 0,C 180,E1 3426.661,E2 3426.661} C_VEL
LIN {X 0,Y 192.563,Z 904.658,A -85,B 0,C 180,E1 3426.1,E2 3426.1} C_VEL
LIN {X 0,Y 199.199,Z 888.392,A -85,B 0,C 180,E1 3425.68,E2 3425.68} C_VEL
LIN {X 0,Y 204.397,Z 870.583,A -85,B 0,C 180,E1 3425.33,E2 3425.33} C_VEL
LIN {X 0,Y 205.206,Z 867.038,A -85,B 0,C 180,E1 3425.251,E2 3425.251} C_VEL
LIN {X 0,Y 200.899,Z 883.08,A -85,B 0,C 180,E1 3424.71,E2 3424.71} C_VEL
LIN {X 0,Y 194.948,Z 898.694,A -85,B 0,C 180,E1 3424.005,E2 3424.005} C_VEL
LIN {X 0,Y 187.066,Z 914.426,A -85,B 0,C 180,E1 3423.063,E2 3423.063} C_VEL
LIN {X 0,Y 178.075,Z 928.596,A -85,B 0,C 180,E1 3421.929,E2 3421.929} C_VEL
LIN {X 0,Y 167.983,Z 941.382,A -85,B 0,C 180,E1 3420.55,E2 3420.55} C_VEL
LIN {X 0,Y 156.017,Z 953.754,A -85,B 0,C 180,E1 3418.699,E2 3418.699} C_VEL
LIN {X 0,Y 143.264,Z 964.53,A -85,B 0,C 180,E1 3416.382,E2 3416.382} C_VEL
LIN {X 0,Y 129.838,Z 973.632,A -85,B 0,C 180,E1 3413.413,E2 3413.413} C_VEL
LIN {X 0,Y 115.915,Z 981.168,A -85,B 0,C 180,E1 3409.524,E2 3409.524} C_VEL
LIN {X 0,Y 102.65,Z 986.732,A -85,B 0,C 180,E1 3404.644,E2 3404.644} C_VEL
LIN {X 0,Y 89.532,Z 990.646,A -85,B 0,C 180,E1 3397.956,E2 3397.956} C_VEL
LIN {X 0,Y 77.872,Z 992.748,A -85,B 0,C 180,E1 3389.095,E2 3389.095} C_VEL
LIN {X 0,Y 68.743,Z 993.071,A -85,B 0,C 180,E1 3377.882,E2 3377.882} C_VEL
LIN {X 0,Y 62.685,Z 991.622,A -85,B 0,C 180,E1 3363.934,E2 3363.934} C_VEL
LIN {X 0,Y 60.527,Z 988.232,A -85,B 0,C 180,E1 3347.296,E2 3347.296} C_VEL
LIN {X 0,Y 62.649,Z 983.229,A -85,B 0,C 180,E1 3331.827,E2 3331.827} C_VEL
LIN {X 0,Y 68.383,Z 976.271,A -85,B 0,C 180,E1 3318.186,E2 3318.186} C_VEL
LIN {X 0,Y 76.373,Z 967.795,A -85,B 0,C 180,E1 3307.686,E2 3307.686} C_VEL
LIN {X 0,Y 85.497,Z 957.711,A -85,B 0,C 180,E1 3299.808,E2 3299.808} C_VEL
LIN {X 0,Y 94.997,Z 946.136,A -85,B 0,C 180,E1 3293.883,E2 3293.883} C_VEL
LIN {X 0,Y 103.964,Z 933.514,A -85,B 0,C 180,E1 3289.519,E2 3289.519} C_VEL
LIN {X 0,Y 112.508,Z 919.201,A -85,B 0,C 180,E1 3286.116,E2 3286.116} C_VEL
LIN {X 0,Y 120.052,Z 903.795,A -85,B 0,C 180,E1 3283.564,E2 3283.564} C_VEL
LIN {X 0,Y 126.274,Z 887.315,A -85,B 0,C 180,E1 3281.66,E2 3281.66} C_VEL
LIN {X 0,Y 131.03,Z 870.165,A -85,B 0,C 180,E1 3280.283,E2 3280.283} C_VEL
LIN {X 0,Y 134.078,Z 852.661,A -85,B 0,C 180,E1 3279.375,E2 3279.375} C_VEL
LIN {X 0,Y 142.456,Z 776.695,A -85,B 0,C 180,E1 3277.146,E2 3277.146} C_VEL
LIN {X 0,Y 142.49,Z 773.278,A -85,B 0,C 180,E1 3276.689,E2 3276.689} C_VEL
LIN {X 0,Y 140.455,Z 766.171,A -85,B 0,C 180,E1 3273.119,E2 3273.119} C_VEL
LIN {X 0,Y 138.845,Z 761.057,A -85,B 0,C 180,E1 3269.677,E2 3269.677} C_VEL
LIN {X 0,Y 137.813,Z 757.938,A -85,B 0,C 180,E1 3266.943,E2 3266.943} C_VEL
LIN {X 0,Y 136.622,Z 754.175,A -85,B 0,C 180,E1 3262.596,E2 3262.596} C_VEL
LIN {X 0,Y 135.929,Z 751.791,A -85,B 0,C 180,E1 3256.232,E2 3256.232} C_VEL
LIN {X 0,Y 136.399,Z 752.19,A -85,B 0,C 180,E1 3250.134,E2 3250.134} C_VEL
LIN {X 0,Y 137.688,Z 754.832,A -85,B 0,C 180,E1 3245,E2 3245} C_VEL
LIN {X 0,Y 139.593,Z 759.153,A -85,B 0,C 180,E1 3240.309,E2 3240.309} C_VEL
LIN {X 0,Y 141.775,Z 764.658,A -85,B 0,C 180,E1 3236.26,E2 3236.26} C_VEL
LIN {X 0,Y 144.549,Z 772.403,A -85,B 0,C 180,E1 3232.149,E2 3232.149} C_VEL
LIN {X 0,Y 144.91,Z 773.918,A -85,B 0,C 180,E1 3231.611,E2 3231.611} C_VEL
LIN {X 0,Y 134.8,Z 866.169,A -85,B 0,C 180,E1 3229.079,E2 3229.079} C_VEL
LIN {X 0,Y 131.039,Z 884.36,A -85,B 0,C 180,E1 3228.191,E2 3228.191} C_VEL
LIN {X 0,Y 125.883,Z 901.055,A -85,B 0,C 180,E1 3227.029,E2 3227.029} C_VEL
LIN {X 0,Y 119.271,Z 917.008,A -85,B 0,C 180,E1 3225.435,E2 3225.435} C_VEL
LIN {X 0,Y 111.113,Z 932.717,A -85,B 0,C 180,E1 3223.122,E2 3223.122} C_VEL
LIN {X 0,Y 101.968,Z 947.355,A -85,B 0,C 180,E1 3219.929,E2 3219.929} C_VEL
LIN {X 0,Y 92.235,Z 960.599,A -85,B 0,C 180,E1 3215.59,E2 3215.59} C_VEL
LIN {X 0,Y 82.278,Z 972.495,A -85,B 0,C 180,E1 3209.637,E2 3209.637} C_VEL
LIN {X 0,Y 72.877,Z 982.955,A -85,B 0,C 180,E1 3201.45,E2 3201.45} C_VEL
LIN {X 0,Y 64.91,Z 991.928,A -85,B 0,C 180,E1 3190.315,E2 3190.315} C_VEL
LIN {X 0,Y 59.716,Z 999.275,A -85,B 0,C 180,E1 3175.809,E2 3175.809} C_VEL
LIN {X 0,Y 58.752,Z 1004.969,A -85,B 0,C 180,E1 3158.812,E2 3158.812} C_VEL
LIN {X 0,Y 60.101,Z 1007.324,A -85,B 0,C 180,E1 3149.049,E2 3149.049} C_VEL
LIN {X 0,Y 58.591,Z 1008.522,A -85,B 0,C 180,E1 3131.083,E2 3131.083} C_VEL
LIN {X 0,Y 63.063,Z 1007.896,A -85,B 0,C 180,E1 3112.953,E2 3112.953} C_VEL
LIN {X 0,Y 72.867,Z 1005.404,A -85,B 0,C 180,E1 3098.545,E2 3098.545} C_VEL
LIN {X 0,Y 85.454,Z 1001.199,A -85,B 0,C 180,E1 3088.655,E2 3088.655} C_VEL
LIN {X 0,Y 100.009,Z 995.106,A -85,B 0,C 180,E1 3081.601,E2 3081.601} C_VEL
LIN {X 0,Y 114.886,Z 987.465,A -85,B 0,C 180,E1 3076.799,E2 3076.799} C_VEL
LIN {X 0,Y 129.523,Z 978.274,A -85,B 0,C 180,E1 3073.43,E2 3073.43} C_VEL
LIN {X 0,Y 143.612,Z 967.57,A -85,B 0,C 180,E1 3070.989,E2 3070.989} C_VEL
LIN {X 0,Y 151.046,Z 961.066,A -85,B 0,C 180,E1 3069.94,E2 3069.94} C_VEL
LIN {X 0,Y 156.235,Z 955.99,A -85,B 0,C 180,E1 3068.907,E2 3068.907} C_VEL
LIN {X 0,Y 167.789,Z 942.489,A -85,B 0,C 180,E1 3065.579,E2 3065.579} C_VEL
LIN {X 0,Y 172.431,Z 936.635,A -85,B 0,C 180,E1 3064.887,E2 3064.887} C_VEL
LIN {X 0,Y 177.834,Z 929.31,A -85,B 0,C 180,E1 3064.514,E2 3064.514} C_VEL
LIN {X 0,Y 167.246,Z 942.472,A -85,B 0,C 180,E1 3063.259,E2 3063.259} C_VEL
LIN {X 0,Y 155.039,Z 954.823,A -85,B 0,C 180,E1 3061.619,E2 3061.619} C_VEL
LIN {X 0,Y 141.983,Z 965.597,A -85,B 0,C 180,E1 3059.561,E2 3059.561} C_VEL
LIN {X 0,Y 128.167,Z 974.714,A -85,B 0,C 180,E1 3056.909,E2 3056.909} C_VEL
LIN {X 0,Y 113.736,Z 982.264,A -85,B 0,C 180,E1 3053.404,E2 3053.404} C_VEL
LIN {X 0,Y 99.838,Z 987.857,A -85,B 0,C 180,E1 3048.942,E2 3048.942} C_VEL
LIN {X 0,Y 85.874,Z 991.806,A -85,B 0,C 180,E1 3042.696,E2 3042.696} C_VEL
LIN {X 0,Y 72.547,Z 994.008,A -85,B 0,C 180,E1 3033.614,E2 3033.614} C_VEL
LIN {X 0,Y 62.248,Z 994.28,A -85,B 0,C 180,E1 3021.91,E2 3021.91} C_VEL
LIN {X 0,Y 55.238,Z 992.78,A -85,B 0,C 180,E1 3006.677,E2 3006.677} C_VEL
LIN {X 0,Y 52.586,Z 989.422,A -85,B 0,C 180,E1 2988.059,E2 2988.059} C_VEL
LIN {X 0,Y 54.652,Z 984.682,A -85,B 0,C 180,E1 2971.046,E2 2971.046} C_VEL
LIN {X 0,Y 60.375,Z 978.298,A -85,B 0,C 180,E1 2956.592,E2 2956.592} C_VEL
LIN {X 0,Y 68.881,Z 970.036,A -85,B 0,C 180,E1 2945.103,E2 2945.103} C_VEL
LIN {X 0,Y 78.567,Z 960.318,A -85,B 0,C 180,E1 2936.821,E2 2936.821} C_VEL
LIN {X 0,Y 88.564,Z 949.05,A -85,B 0,C 180,E1 2930.784,E2 2930.784} C_VEL
LIN {X 0,Y 98.369,Z 936.29,A -85,B 0,C 180,E1 2926.275,E2 2926.275} C_VEL
LIN {X 0,Y 107.265,Z 922.462,A -85,B 0,C 180,E1 2922.967,E2 2922.967} C_VEL
LIN {X 0,Y 115.525,Z 906.692,A -85,B 0,C 180,E1 2920.39,E2 2920.39} C_VEL
LIN {X 0,Y 121.668,Z 891.885,A -85,B 0,C 180,E1 2918.673,E2 2918.673} C_VEL
LIN {X 0,Y 126.848,Z 875.082,A -85,B 0,C 180,E1 2917.307,E2 2917.307} C_VEL
LIN {X 0,Y 130.526,Z 857.342,A -85,B 0,C 180,E1 2916.337,E2 2916.337} C_VEL
LIN {X 0,Y 137.323,Z 798.92,A -85,B 0,C 180,E1 2914.696,E2 2914.696} C_VEL
LIN {X 0,Y 139.673,Z 777.762,A -85,B 0,C 180,E1 2914.103,E2 2914.103} C_VEL
LIN {X 0,Y 137.837,Z 770.45,A -85,B 0,C 180,E1 2910.036,E2 2910.036} C_VEL
LIN {X 0,Y 136.44,Z 765.567,A -85,B 0,C 180,E1 2906.085,E2 2906.085} C_VEL
LIN {X 0,Y 135.402,Z 761.828,A -85,B 0,C 180,E1 2901.668,E2 2901.668} C_VEL
LIN {X 0,Y 134.927,Z 759.714,A -85,B 0,C 180,E1 2895.914,E2 2895.914} C_VEL
LIN {X 0,Y 135.375,Z 760.176,A -85,B 0,C 180,E1 2890.211,E2 2890.211} C_VEL
LIN {X 0,Y 136.415,Z 762.628,A -85,B 0,C 180,E1 2885.679,E2 2885.679} C_VEL
LIN {X 0,Y 137.978,Z 766.511,A -85,B 0,C 180,E1 2881.433,E2 2881.433} C_VEL
LIN {X 0,Y 139.943,Z 772.105,A -85,B 0,C 180,E1 2877.339,E2 2877.339} C_VEL
LIN {X 0,Y 141.573,Z 777.572,A -85,B 0,C 180,E1 2874.499,E2 2874.499} C_VEL
LIN {X 0,Y 131.597,Z 865.607,A -85,B 0,C 180,E1 2872.237,E2 2872.237} C_VEL
LIN {X 0,Y 127.715,Z 883.804,A -85,B 0,C 180,E1 2871.416,E2 2871.416} C_VEL
LIN {X 0,Y 122.227,Z 900.984,A -85,B 0,C 180,E1 2870.316,E2 2870.316} C_VEL
LIN {X 0,Y 115.18,Z 917.254,A -85,B 0,C 180,E1 2868.802,E2 2868.802} C_VEL
LIN {X 0,Y 106.403,Z 933.379,A -85,B 0,C 180,E1 2866.558,E2 2866.558} C_VEL
LIN {X 0,Y 96.96,Z 947.661,A -85,B 0,C 180,E1 2863.546,E2 2863.546} C_VEL
LIN {X 0,Y 86.597,Z 960.861,A -85,B 0,C 180,E1 2859.27,E2 2859.27} C_VEL
LIN {X 0,Y 76.08,Z 972.56,A -85,B 0,C 180,E1 2853.342,E2 2853.342} C_VEL
LIN {X 0,Y 65.946,Z 982.885,A -85,B 0,C 180,E1 2844.822,E2 2844.822} C_VEL
LIN {X 0,Y 57.354,Z 991.538,A -85,B 0,C 180,E1 2832.838,E2 2832.838} C_VEL
LIN {X 0,Y 51.721,Z 998.712,A -85,B 0,C 180,E1 2816.402,E2 2816.402} C_VEL
LIN {X 0,Y 50.862,Z 1003.956,A -85,B 0,C 180,E1 2797.912,E2 2797.912} C_VEL
LIN {X 0,Y 52.004,Z 1005.877,A -85,B 0,C 180,E1 2788.702,E2 2788.702} C_VEL
LIN {X 0,Y 50.935,Z 1007.193,A -85,B 0,C 180,E1 2768.103,E2 2768.103} C_VEL
LIN {X 0,Y 56.73,Z 1006.676,A -85,B 0,C 180,E1 2747.955,E2 2747.955} C_VEL
LIN {X 0,Y 68.051,Z 1004.299,A -85,B 0,C 180,E1 2733.127,E2 2733.127} C_VEL
LIN {X 0,Y 81.833,Z 1000.261,A -85,B 0,C 180,E1 2723.602,E2 2723.602} C_VEL
LIN {X 0,Y 97.292,Z 994.282,A -85,B 0,C 180,E1 2717.111,E2 2717.111} C_VEL
LIN {X 0,Y 113.027,Z 986.647,A -85,B 0,C 180,E1 2712.776,E2 2712.776} C_VEL
LIN {X 0,Y 127.879,Z 977.781,A -85,B 0,C 180,E1 2709.884,E2 2709.884} C_VEL
LIN {X 0,Y 142.291,Z 967.22,A -85,B 0,C 180,E1 2707.787,E2 2707.787} C_VEL
LIN {X 0,Y 156.147,Z 954.898,A -85,B 0,C 180,E1 2706.249,E2 2706.249} C_VEL
LIN {X 0,Y 168.168,Z 941.934,A -85,B 0,C 180,E1 2705.203,E2 2705.203} C_VEL
LIN {X 0,Y 172.431,Z 936.635,A -85,B 0,C 180,E1 2704.887,E2 2704.887} C_VEL
LIN {X 0,Y 171.155,Z 938.112,A -85,B 0,C 180,E1 2704.561,E2 2704.561} C_VEL
LIN {X 0,Y 164.055,Z 946.249,A -85,B 0,C 180,E1 2704.155,E2 2704.155} C_VEL
LIN {X 0,Y 152.241,Z 957.885,A -85,B 0,C 180,E1 2704.073,E2 2704.073} C_VEL
LIN {X 0,Y 142.842,Z 965.804,A -85,B 0,C 180,E1 2704.439,E2 2704.439} C_VEL
LIN {X 0,Y 139.619,Z 968.257,A -85,B 0,C 180,E1 2704.722,E2 2704.722} C_VEL
LIN {X 0,Y 124.791,Z 978.444,A -85,B 0,C 180,E1 2706.53,E2 2706.53} C_VEL
LIN {X 0,Y 109.358,Z 987.078,A -85,B 0,C 180,E1 2709.095,E2 2709.095} C_VEL
LIN {X 0,Y 93.35,Z 994.239,A -85,B 0,C 180,E1 2712.923,E2 2712.923} C_VEL
LIN {X 0,Y 77.162,Z 999.788,A -85,B 0,C 180,E1 2718.93,E2 2718.93} C_VEL
LIN {X 0,Y 61.638,Z 1003.69,A -85,B 0,C 180,E1 2728.844,E2 2728.844} C_VEL
LIN {X 0,Y 49.827,Z 1005.608,A -85,B 0,C 180,E1 2743.75,E2 2743.75} C_VEL
LIN {X 0,Y 43.142,Z 1005.734,A -85,B 0,C 180,E1 2766.799,E2 2766.799} C_VEL
LIN {X 0,Y 43.996,Z 1004.283,A -85,B 0,C 180,E1 2789.235,E2 2789.235} C_VEL
LIN {X 0,Y 43.018,Z 999.572,A -85,B 0,C 180,E1 2811.835,E2 2811.835} C_VEL
LIN {X 0,Y 47.941,Z 993.107,A -85,B 0,C 180,E1 2831.87,E2 2831.87} C_VEL
LIN {X 0,Y 56.641,Z 985.074,A -85,B 0,C 180,E1 2846.068,E2 2846.068} C_VEL
LIN {X 0,Y 67.82,Z 974.869,A -85,B 0,C 180,E1 2856.078,E2 2856.078} C_VEL
LIN {X 0,Y 78.735,Z 963.949,A -85,B 0,C 180,E1 2862.262,E2 2862.262} C_VEL
LIN {X 0,Y 89.44,Z 951.638,A -85,B 0,C 180,E1 2866.557,E2 2866.557} C_VEL
LIN {X 0,Y 99.61,Z 937.757,A -85,B 0,C 180,E1 2869.648,E2 2869.648} C_VEL
LIN {X 0,Y 108.597,Z 923.005,A -85,B 0,C 180,E1 2871.801,E2 2871.801} C_VEL
LIN {X 0,Y 116.277,Z 907.457,A -85,B 0,C 180,E1 2873.312,E2 2873.312} C_VEL
LIN {X 0,Y 122.569,Z 890.788,A -85,B 0,C 180,E1 2874.405,E2 2874.405} C_VEL
LIN {X 0,Y 127.357,Z 872.766,A -85,B 0,C 180,E1 2875.264,E2 2875.264} C_VEL
LIN {X 0,Y 130.235,Z 854.846,A -85,B 0,C 180,E1 2875.83,E2 2875.83} C_VEL
LIN {X 0,Y 138.611,Z 781.237,A -85,B 0,C 180,E1 2877.52,E2 2877.52} C_VEL
LIN {X 0,Y 136.791,Z 775.121,A -85,B 0,C 180,E1 2881.572,E2 2881.572} C_VEL
LIN {X 0,Y 135.595,Z 771.677,A -85,B 0,C 180,E1 2884.865,E2 2884.865} C_VEL
LIN {X 0,Y 134.743,Z 769.256,A -85,B 0,C 180,E1 2888.106,E2 2888.106} C_VEL
LIN {X 0,Y 134.165,Z 767.841,A -85,B 0,C 180,E1 2891.609,E2 2891.609} C_VEL
LIN {X 0,Y 133.926,Z 767.773,A -85,B 0,C 180,E1 2896.482,E2 2896.482} C_VEL
LIN {X 0,Y 134.391,Z 770.161,A -85,B 0,C 180,E1 2901.84,E2 2901.84} C_VEL
LIN {X 0,Y 135.393,Z 774.493,A -85,B 0,C 180,E1 2906.302,E2 2906.302} C_VEL
LIN {X 0,Y 136.511,Z 779.372,A -85,B 0,C 180,E1 2909.752,E2 2909.752} C_VEL
LIN {X 0,Y 136.997,Z 781.975,A -85,B 0,C 180,E1 2911.118,E2 2911.118} C_VEL
LIN {X 0,Y 128.175,Z 856.513,A -85,B 0,C 180,E1 2912.931,E2 2912.931} C_VEL
LIN {X 0,Y 124.637,Z 873.841,A -85,B 0,C 180,E1 2913.766,E2 2913.766} C_VEL
LIN {X 0,Y 119.546,Z 890.452,A -85,B 0,C 180,E1 2914.948,E2 2914.948} C_VEL
LIN {X 0,Y 113.195,Z 905.867,A -85,B 0,C 180,E1 2916.502,E2 2916.502} C_VEL
LIN {X 0,Y 105.06,Z 921.191,A -85,B 0,C 180,E1 2918.701,E2 2918.701} C_VEL
LIN {X 0,Y 95.745,Z 935.477,A -85,B 0,C 180,E1 2921.695,E2 2921.695} C_VEL
LIN {X 0,Y 85.808,Z 948.096,A -85,B 0,C 180,E1 2925.64,E2 2925.64} C_VEL
LIN {X 0,Y 75.05,Z 959.692,A -85,B 0,C 180,E1 2931.23,E2 2931.23} C_VEL
LIN {X 0,Y 64.374,Z 969.815,A -85,B 0,C 180,E1 2939.163,E2 2939.163} C_VEL
LIN {X 0,Y 54.609,Z 978.344,A -85,B 0,C 180,E1 2950.755,E2 2950.755} C_VEL
LIN {X 0,Y 47.278,Z 985.363,A -85,B 0,C 180,E1 2967.574,E2 2967.574} C_VEL
LIN {X 0,Y 44.651,Z 990.211,A -85,B 0,C 180,E1 2986.922,E2 2986.922} C_VEL
LIN {X 0,Y 47.248,Z 993.625,A -85,B 0,C 180,E1 3007.855,E2 3007.855} C_VEL
LIN {X 0,Y 55.626,Z 995.431,A -85,B 0,C 180,E1 3026.134,E2 3026.134} C_VEL
LIN {X 0,Y 66.821,Z 995.365,A -85,B 0,C 180,E1 3038.079,E2 3038.079} C_VEL
LIN {X 0,Y 80.192,Z 993.508,A -85,B 0,C 180,E1 3046.536,E2 3046.536} C_VEL
LIN {X 0,Y 95.517,Z 989.632,A -85,B 0,C 180,E1 3052.783,E2 3052.783} C_VEL
LIN {X 0,Y 110.14,Z 984.249,A -85,B 0,C 180,E1 3056.941,E2 3056.941} C_VEL
LIN {X 0,Y 124.981,Z 976.924,A -85,B 0,C 180,E1 3060.113,E2 3060.113} C_VEL
LIN {X 0,Y 139.11,Z 968.094,A -85,B 0,C 180,E1 3062.487,E2 3062.487} C_VEL
LIN {X 0,Y 148.63,Z 960.926,A -85,B 0,C 180,E1 3063.857,E2 3063.857} C_VEL
LIN {X 0,Y 139.619,Z 968.257,A -85,B 0,C 180,E1 3064.722,E2 3064.722} C_VEL
LIN {X 0,Y 134.147,Z 972.181,A -85,B 0,C 180,E1 3064.946,E2 3064.946} C_VEL
LIN {X 0,Y 126.565,Z 976.839,A -85,B 0,C 180,E1 3064.393,E2 3064.393} C_VEL
LIN {X 0,Y 114.936,Z 982.781,A -85,B 0,C 180,E1 3062.355,E2 3062.355} C_VEL
LIN {X 0,Y 109.037,Z 985.343,A -85,B 0,C 180,E1 3061.127,E2 3061.127} C_VEL
LIN {X 0,Y 93.765,Z 990.788,A -85,B 0,C 180,E1 3057.554,E2 3057.554} C_VEL
LIN {X 0,Y 78.654,Z 994.492,A -85,B 0,C 180,E1 3052.535,E2 3052.535} C_VEL
LIN {X 0,Y 64.143,Z 996.483,A -85,B 0,C 180,E1 3045.112,E2 3045.112} C_VEL
LIN {X 0,Y 51.252,Z 996.739,A -85,B 0,C 180,E1 3033.815,E2 3033.815} C_VEL
LIN {X 0,Y 41.393,Z 995.233,A -85,B 0,C 180,E1 3016.437,E2 3016.437} C_VEL
LIN {X 0,Y 36.744,Z 991.807,A -85,B 0,C 180,E1 2990.714,E2 2990.714} C_VEL
LIN {X 0,Y 39.374,Z 986.799,A -85,B 0,C 180,E1 2965.628,E2 2965.628} C_VEL
LIN {X 0,Y 47.567,Z 979.857,A -85,B 0,C 180,E1 2946.458,E2 2946.458} C_VEL
LIN {X 0,Y 58.284,Z 971.435,A -85,B 0,C 180,E1 2934.317,E2 2934.317} C_VEL
LIN {X 0,Y 69.739,Z 961.478,A -85,B 0,C 180,E1 2926.511,E2 2926.511} C_VEL
LIN {X 0,Y 81.093,Z 950.037,A -85,B 0,C 180,E1 2921.223,E2 2921.223} C_VEL
LIN {X 0,Y 91.935,Z 937.08,A -85,B 0,C 180,E1 2917.444,E2 2917.444} C_VEL
LIN {X 0,Y 101.602,Z 922.941,A -85,B 0,C 180,E1 2914.74,E2 2914.74} C_VEL
LIN {X 0,Y 109.999,Z 907.817,A -85,B 0,C 180,E1 2912.773,E2 2912.773} C_VEL
LIN {X 0,Y 116.546,Z 892.855,A -85,B 0,C 180,E1 2911.39,E2 2911.39} C_VEL
LIN {X 0,Y 122.077,Z 875.725,A -85,B 0,C 180,E1 2910.277,E2 2910.277} C_VEL
LIN {X 0,Y 125.907,Z 858.061,A -85,B 0,C 180,E1 2909.494,E2 2909.494} C_VEL
LIN {X 0,Y 133.799,Z 793.284,A -85,B 0,C 180,E1 2908.045,E2 2908.045} C_VEL
LIN {X 0,Y 134.687,Z 785.799,A -85,B 0,C 180,E1 2907.885,E2 2907.885} C_VEL
LIN {X 0,Y 133.759,Z 780.779,A -85,B 0,C 180,E1 2904.219,E2 2904.219} C_VEL
LIN {X 0,Y 133.117,Z 777.288,A -85,B 0,C 180,E1 2900.131,E2 2900.131} C_VEL
LIN {X 0,Y 132.934,Z 775.569,A -85,B 0,C 180,E1 2895.264,E2 2895.264} C_VEL
LIN {X 0,Y 133.277,Z 776.135,A -85,B 0,C 180,E1 2890.642,E2 2890.642} C_VEL
LIN {X 0,Y 133.879,Z 778.024,A -85,B 0,C 180,E1 2887.295,E2 2887.295} C_VEL
LIN {X 0,Y 134.88,Z 781.316,A -85,B 0,C 180,E1 2883.72,E2 2883.72} C_VEL
LIN {X 0,Y 135.976,Z 785.54,A -85,B 0,C 180,E1 2880.647,E2 2880.647} C_VEL
LIN {X 0,Y 126.484,Z 864.422,A -85,B 0,C 180,E1 2878.983,E2 2878.983} C_VEL
LIN {X 0,Y 122.35,Z 882.766,A -85,B 0,C 180,E1 2878.332,E2 2878.332} C_VEL
LIN {X 0,Y 116.646,Z 899.723,A -85,B 0,C 180,E1 2877.509,E2 2877.509} C_VEL
LIN {X 0,Y 109.205,Z 916.001,A -85,B 0,C 180,E1 2876.381,E2 2876.381} C_VEL
LIN {X 0,Y 100.405,Z 931.263,A -85,B 0,C 180,E1 2874.778,E2 2874.778} C_VEL
LIN {X 0,Y 90.225,Z 945.662,A -85,B 0,C 180,E1 2872.435,E2 2872.435} C_VEL
LIN {X 0,Y 79.177,Z 958.569,A -85,B 0,C 180,E1 2869.082,E2 2869.082} C_VEL
LIN {X 0,Y 67.551,Z 970.097,A -85,B 0,C 180,E1 2864.184,E2 2864.184} C_VEL
LIN {X 0,Y 55.641,Z 980.427,A -85,B 0,C 180,E1 2856.42,E2 2856.42} C_VEL
LIN {X 0,Y 44.623,Z 989.193,A -85,B 0,C 180,E1 2843.774,E2 2843.774} C_VEL
LIN {X 0,Y 36.62,Z 996.386,A -85,B 0,C 180,E1 2823.101,E2 2823.101} C_VEL
LIN {X 0,Y 35.008,Z 1001.63,A -85,B 0,C 180,E1 2796.563,E2 2796.563} C_VEL
LIN {X 0,Y 35.917,Z 1002.85,A -85,B 0,C 180,E1 2788.408,E2 2788.408} C_VEL
LIN {X 0,Y 36.3,Z 1004.433,A -85,B 0,C 180,E1 2758.447,E2 2758.447} C_VEL
LIN {X 0,Y 45.881,Z 1004.239,A -85,B 0,C 180,E1 2734.098,E2 2734.098} C_VEL
